LIN {X 0,Y 256.06,Z 399.2,A -85,B 0,C 180,E1 -18513.951,E2 -18513.951} C_VEL
LIN {X 0,Y 256.043,Z 399.215,A -85,B 0,C 180,E1 -18517.401,E2 -18517.401} C_VEL
LIN {X 0,Y 256.093,Z 399.188,A -85,B 0,C 180,E1 -18520.773,E2 -18520.773} C_VEL
LIN {X 0,Y 256.198,Z 399.177,A -85,B 0,C 180,E1 -18524.079,E2 -18524.079} C_VEL
LIN {X 0,Y 256.273,Z 399.171,A -85,B 0,C 180,E1 -18528.933,E2 -18528.933} C_VEL
LIN {X 0,Y 256.453,Z 399.151,A -85,B 0,C 180,E1 -18532.125,E2 -18532.125} C_VEL
LIN {X 0,Y 256.439,Z 399.144,A -85,B 0,C 180,E1 -18536.858,E2 -18536.858} C_VEL
LIN {X 0,Y 256.682,Z 399.137,A -85,B 0,C 180,E1 -18538.431,E2 -18538.431} C_VEL
LIN {X 0,Y 256.686,Z 399.109,A -85,B 0,C 180,E1 -18541.569,E2 -18541.569} C_VEL
LIN {X 0,Y 256.436,Z 399.14,A -85,B 0,C 180,E1 -18546.787,E2 -18546.787} C_VEL
LIN {X 0,Y 256.388,Z 399.171,A -85,B 0,C 180,E1 -18549.467,E2 -18549.467} C_VEL
LIN {X 0,Y 256.219,Z 399.192,A -85,B 0,C 180,E1 -18554.292,E2 -18554.292} C_VEL
LIN {X 0,Y 256.149,Z 399.182,A -85,B 0,C 180,E1 -18557.566,E2 -18557.566} C_VEL
LIN {X 0,Y 256.106,Z 399.186,A -85,B 0,C 180,E1 -18561.098,E2 -18561.098} C_VEL
LIN {X 0,Y 256.084,Z 399.409,A -85,B 0,C 180,E1 -18564.094,E2 -18564.094} C_VEL
LIN {X 0,Y 256.517,Z 400.923,A -85,B 0,C 180,E1 -18564.875,E2 -18564.875} C_VEL
LIN {X 0,Y 258.666,Z 404.243,A -85,B 0,C 180,E1 -18566.635,E2 -18566.635} C_VEL
LIN {X 0,Y 259.435,Z 406.128,A -85,B 0,C 180,E1 -18567.421,E2 -18567.421} C_VEL
LIN {X 0,Y 260.409,Z 407.557,A -85,B 0,C 180,E1 -18568.184,E2 -18568.184} C_VEL
LIN {X 0,Y 264.822,Z 416.275,A -85,B 0,C 180,E1 -18571.877,E2 -18571.877} C_VEL
LIN {X 0,Y 268.116,Z 423.333,A -85,B 0,C 180,E1 -18574.513,E2 -18574.513} C_VEL
LIN {X 0,Y 272.289,Z 433.348,A -85,B 0,C 180,E1 -18577.807,E2 -18577.807} C_VEL
LIN {X 0,Y 275.747,Z 442.564,A -85,B 0,C 180,E1 -18580.535,E2 -18580.535} C_VEL
LIN {X 0,Y 279.195,Z 452.902,A -85,B 0,C 180,E1 -18583.309,E2 -18583.309} C_VEL
LIN {X 0,Y 282.851,Z 466.067,A -85,B 0,C 180,E1 -18586.453,E2 -18586.453} C_VEL
LIN {X 0,Y 284.238,Z 471.069,A -85,B 0,C 180,E1 -18587.467,E2 -18587.467} C_VEL
LIN {X 0,Y 285.594,Z 474.475,A -85,B 0,C 180,E1 -18587.831,E2 -18587.831} C_VEL
LIN {X 0,Y 289.442,Z 502.295,A -85,B 0,C 180,E1 -18589.411,E2 -18589.411} C_VEL
LIN {X 0,Y 291.695,Z 522.529,A -85,B 0,C 180,E1 -18590.425,E2 -18590.425} C_VEL
LIN {X 0,Y 286.727,Z 629.994,A -85,B 0,C 180,E1 -18592.986,E2 -18592.986} C_VEL
LIN {X 0,Y 285.652,Z 646.755,A -85,B 0,C 180,E1 -18593.484,E2 -18593.484} C_VEL
LIN {X 0,Y 283.945,Z 662.444,A -85,B 0,C 180,E1 -18594.218,E2 -18594.218} C_VEL
LIN {X 0,Y 281.63,Z 677.308,A -85,B 0,C 180,E1 -18595.186,E2 -18595.186} C_VEL
LIN {X 0,Y 279.166,Z 690.887,A -85,B 0,C 180,E1 -18596.372,E2 -18596.372} C_VEL
LIN {X 0,Y 276.125,Z 704.824,A -85,B 0,C 180,E1 -18597.909,E2 -18597.909} C_VEL
LIN {X 0,Y 272.866,Z 717.487,A -85,B 0,C 180,E1 -18599.641,E2 -18599.641} C_VEL
LIN {X 0,Y 269.642,Z 729.09,A -85,B 0,C 180,E1 -18601.6,E2 -18601.6} C_VEL
LIN {X 0,Y 266.466,Z 740.121,A -85,B 0,C 180,E1 -18603.888,E2 -18603.888} C_VEL
LIN {X 0,Y 263.832,Z 748.759,A -85,B 0,C 180,E1 -18606.035,E2 -18606.035} C_VEL
LIN {X 0,Y 260.992,Z 757.604,A -85,B 0,C 180,E1 -18608.686,E2 -18608.686} C_VEL
LIN {X 0,Y 258.674,Z 765.048,A -85,B 0,C 180,E1 -18611.427,E2 -18611.427} C_VEL
LIN {X 0,Y 256.961,Z 770.984,A -85,B 0,C 180,E1 -18614.13,E2 -18614.13} C_VEL
LIN {X 0,Y 255.426,Z 776.513,A -85,B 0,C 180,E1 -18617.287,E2 -18617.287} C_VEL
LIN {X 0,Y 254.539,Z 780.689,A -85,B 0,C 180,E1 -18620.467,E2 -18620.467} C_VEL
LIN {X 0,Y 254.052,Z 783.623,A -85,B 0,C 180,E1 -18623.65,E2 -18623.65} C_VEL
LIN {X 0,Y 253.901,Z 785.384,A -85,B 0,C 180,E1 -18626.829,E2 -18626.829} C_VEL
LIN {X 0,Y 253.945,Z 785.994,A -85,B 0,C 180,E1 -18630.002,E2 -18630.002} C_VEL
LIN {X 0,Y 253.904,Z 785.421,A -85,B 0,C 180,E1 -18633.176,E2 -18633.176} C_VEL
LIN {X 0,Y 254.057,Z 783.708,A -85,B 0,C 180,E1 -18636.355,E2 -18636.355} C_VEL
LIN {X 0,Y 254.539,Z 780.819,A -85,B 0,C 180,E1 -18639.538,E2 -18639.538} C_VEL
LIN {X 0,Y 255.402,Z 776.687,A -85,B 0,C 180,E1 -18642.72,E2 -18642.72} C_VEL
LIN {X 0,Y 256.911,Z 771.213,A -85,B 0,C 180,E1 -18645.878,E2 -18645.878} C_VEL
LIN {X 0,Y 258.919,Z 764.244,A -85,B 0,C 180,E1 -18649.012,E2 -18649.012} C_VEL
LIN {X 0,Y 261.267,Z 756.773,A -85,B 0,C 180,E1 -18651.71,E2 -18651.71} C_VEL
LIN {X 0,Y 264.2,Z 747.772,A -85,B 0,C 180,E1 -18654.353,E2 -18654.353} C_VEL
LIN {X 0,Y 266.946,Z 738.581,A -85,B 0,C 180,E1 -18656.59,E2 -18656.59} C_VEL
LIN {X 0,Y 270.134,Z 727.708,A -85,B 0,C 180,E1 -18658.773,E2 -18658.773} C_VEL
LIN {X 0,Y 273.395,Z 715.822,A -85,B 0,C 180,E1 -18660.727,E2 -18660.727} C_VEL
LIN {X 0,Y 276.662,Z 702.814,A -85,B 0,C 180,E1 -18662.457,E2 -18662.457} C_VEL
LIN {X 0,Y 279.56,Z 689.399,A -85,B 0,C 180,E1 -18663.889,E2 -18663.889} C_VEL
LIN {X 0,Y 282.042,Z 675.326,A -85,B 0,C 180,E1 -18665.079,E2 -18665.079} C_VEL
LIN {X 0,Y 284.262,Z 660.41,A -85,B 0,C 180,E1 -18666.015,E2 -18666.015} C_VEL
LIN {X 0,Y 285.929,Z 644.861,A -85,B 0,C 180,E1 -18666.7,E2 -18666.7} C_VEL
LIN {X 0,Y 286.971,Z 626.833,A -85,B 0,C 180,E1 -18667.203,E2 -18667.203} C_VEL
LIN {X 0,Y 291.838,Z 522.454,A -85,B 0,C 180,E1 -18669.684,E2 -18669.684} C_VEL
LIN {X 0,Y 288.761,Z 496.622,A -85,B 0,C 180,E1 -18671.019,E2 -18671.019} C_VEL
LIN {X 0,Y 285.637,Z 474.073,A -85,B 0,C 180,E1 -18672.309,E2 -18672.309} C_VEL
LIN {X 0,Y 283.934,Z 470.142,A -85,B 0,C 180,E1 -18672.808,E2 -18672.808} C_VEL
LIN {X 0,Y 280.783,Z 458.187,A -85,B 0,C 180,E1 -18675.505,E2 -18675.505} C_VEL
LIN {X 0,Y 276.887,Z 445.879,A -85,B 0,C 180,E1 -18678.705,E2 -18678.705} C_VEL
LIN {X 0,Y 273.015,Z 434.978,A -85,B 0,C 180,E1 -18681.843,E2 -18681.843} C_VEL
LIN {X 0,Y 270.59,Z 428.968,A -85,B 0,C 180,E1 -18683.781,E2 -18683.781} C_VEL
LIN {X 0,Y 268.817,Z 426.664,A -85,B 0,C 180,E1 -18684.753,E2 -18684.753} C_VEL
LIN {X 0,Y 266.276,Z 425.384,A -85,B 0,C 180,E1 -18685.747,E2 -18685.747} C_VEL
LIN {X 0,Y 262.402,Z 425.077,A -85,B 0,C 180,E1 -18686.98,E2 -18686.98} C_VEL
LIN {X 0,Y 259.868,Z 425.572,A -85,B 0,C 180,E1 -18687.69,E2 -18687.69} C_VEL
LIN {X 0,Y 259.216,Z 426.104,A -85,B 0,C 180,E1 -18688.054,E2 -18688.054} C_VEL
LIN {X 0,Y 259.503,Z 427.426,A -85,B 0,C 180,E1 -18688.288,E2 -18688.288} C_VEL
LIN {X 0,Y 264.767,Z 441.663,A -85,B 0,C 180,E1 -18689.367,E2 -18689.367} C_VEL
LIN {X 0,Y 259.318,Z 542.125,A -85,B 0,C 180,E1 -18693.539,E2 -18693.539} C_VEL
LIN {X 0,Y 258.632,Z 557.649,A -85,B 0,C 180,E1 -18694.39,E2 -18694.39} C_VEL
LIN {X 0,Y 257.663,Z 572.895,A -85,B 0,C 180,E1 -18695.527,E2 -18695.527} C_VEL
LIN {X 0,Y 256.55,Z 586.386,A -85,B 0,C 180,E1 -18696.809,E2 -18696.809} C_VEL
LIN {X 0,Y 255.232,Z 601.418,A -85,B 0,C 180,E1 -18698.602,E2 -18698.602} C_VEL
LIN {X 0,Y 253.81,Z 615.052,A -85,B 0,C 180,E1 -18700.593,E2 -18700.593} C_VEL
LIN {X 0,Y 252.583,Z 627.546,A -85,B 0,C 180,E1 -18702.804,E2 -18702.804} C_VEL
LIN {X 0,Y 251.52,Z 637.995,A -85,B 0,C 180,E1 -18705.021,E2 -18705.021} C_VEL
LIN {X 0,Y 250.66,Z 647.631,A -85,B 0,C 180,E1 -18707.45,E2 -18707.45} C_VEL
LIN {X 0,Y 249.954,Z 656.985,A -85,B 0,C 180,E1 -18710.287,E2 -18710.287} C_VEL
LIN {X 0,Y 249.49,Z 663.619,A -85,B 0,C 180,E1 -18712.717,E2 -18712.717} C_VEL
LIN {X 0,Y 249.243,Z 670.808,A -85,B 0,C 180,E1 -18715.958,E2 -18715.958} C_VEL
LIN {X 0,Y 249.469,Z 676.374,A -85,B 0,C 180,E1 -18719.193,E2 -18719.193} C_VEL
LIN {X 0,Y 250.022,Z 679.487,A -85,B 0,C 180,E1 -18721.611,E2 -18721.611} C_VEL
LIN {X 0,Y 251.132,Z 682.416,A -85,B 0,C 180,E1 -18724.816,E2 -18724.816} C_VEL
LIN {X 0,Y 252.623,Z 684.009,A -85,B 0,C 180,E1 -18727.996,E2 -18727.996} C_VEL
LIN {X 0,Y 254.788,Z 684.233,A -85,B 0,C 180,E1 -18731.133,E2 -18731.133} C_VEL
LIN {X 0,Y 257.49,Z 683.132,A -85,B 0,C 180,E1 -18734.22,E2 -18734.22} C_VEL
LIN {X 0,Y 260.989,Z 680.652,A -85,B 0,C 180,E1 -18737.23,E2 -18737.23} C_VEL
LIN {X 0,Y 264.933,Z 676.843,A -85,B 0,C 180,E1 -18740.173,E2 -18740.173} C_VEL
LIN {X 0,Y 269.585,Z 671.523,A -85,B 0,C 180,E1 -18743.019,E2 -18743.019} C_VEL
LIN {X 0,Y 274.771,Z 664.681,A -85,B 0,C 180,E1 -18745.774,E2 -18745.774} C_VEL
LIN {X 0,Y 279.832,Z 657.27,A -85,B 0,C 180,E1 -18748.093,E2 -18748.093} C_VEL
LIN {X 0,Y 286.156,Z 647.005,A -85,B 0,C 180,E1 -18750.638,E2 -18750.638} C_VEL
LIN {X 0,Y 292.113,Z 636.101,A -85,B 0,C 180,E1 -18752.774,E2 -18752.774} C_VEL
LIN {X 0,Y 298.05,Z 624.066,A -85,B 0,C 180,E1 -18754.671,E2 -18754.671} C_VEL
LIN {X 0,Y 302.909,Z 613.048,A -85,B 0,C 180,E1 -18756.068,E2 -18756.068} C_VEL
LIN {X 0,Y 308.468,Z 598.622,A -85,B 0,C 180,E1 -18757.55,E2 -18757.55} C_VEL
LIN {X 0,Y 312.634,Z 585.97,A -85,B 0,C 180,E1 -18758.595,E2 -18758.595} C_VEL
LIN {X 0,Y 317.001,Z 569.833,A -85,B 0,C 180,E1 -18759.649,E2 -18759.649} C_VEL
LIN {X 0,Y 321.934,Z 549.906,A -85,B 0,C 180,E1 -18760.655,E2 -18760.655} C_VEL
LIN {X 0,Y 331.491,Z 513.679,A -85,B 0,C 180,E1 -18762.202,E2 -18762.202} C_VEL
LIN {X 0,Y 331.324,Z 514.505,A -85,B 0,C 180,E1 -18763.011,E2 -18763.011} C_VEL
LIN {X 0,Y 328.78,Z 524.894,A -85,B 0,C 180,E1 -18763.854,E2 -18763.854} C_VEL
LIN {X 0,Y 327.692,Z 529.255,A -85,B 0,C 180,E1 -18764.081,E2 -18764.081} C_VEL
LIN {X 0,Y 312.213,Z 593.031,A -85,B 0,C 180,E1 -18766.639,E2 -18766.639} C_VEL
LIN {X 0,Y 306.727,Z 610.777,A -85,B 0,C 180,E1 -18767.503,E2 -18767.503} C_VEL
LIN {X 0,Y 300.345,Z 628.134,A -85,B 0,C 180,E1 -18768.618,E2 -18768.618} C_VEL
LIN {X 0,Y 293.51,Z 644.352,A -85,B 0,C 180,E1 -18769.944,E2 -18769.944} C_VEL
LIN {X 0,Y 286.435,Z 659.292,A -85,B 0,C 180,E1 -18771.491,E2 -18771.491} C_VEL
LIN {X 0,Y 279.486,Z 673.037,A -85,B 0,C 180,E1 -18773.327,E2 -18773.327} C_VEL
LIN {X 0,Y 274.434,Z 683.089,A -85,B 0,C 180,E1 -18774.938,E2 -18774.938} C_VEL
LIN {X 0,Y 271.434,Z 697.667,A -85,B 0,C 180,E1 -18776.394,E2 -18776.394} C_VEL
LIN {X 0,Y 268.34,Z 710.262,A -85,B 0,C 180,E1 -18777.968,E2 -18777.968} C_VEL
LIN {X 0,Y 264.895,Z 722.987,A -85,B 0,C 180,E1 -18779.946,E2 -18779.946} C_VEL
LIN {X 0,Y 261.612,Z 733.628,A -85,B 0,C 180,E1 -18781.955,E2 -18781.955} C_VEL
LIN {X 0,Y 258.634,Z 743.458,A -85,B 0,C 180,E1 -18784.227,E2 -18784.227} C_VEL
LIN {X 0,Y 255.453,Z 753.06,A -85,B 0,C 180,E1 -18786.916,E2 -18786.916} C_VEL
LIN {X 0,Y 252.869,Z 761.05,A -85,B 0,C 180,E1 -18789.669,E2 -18789.669} C_VEL
LIN {X 0,Y 250.628,Z 768.04,A -85,B 0,C 180,E1 -18792.642,E2 -18792.642} C_VEL
LIN {X 0,Y 248.854,Z 774.37,A -85,B 0,C 180,E1 -18796.108,E2 -18796.108} C_VEL
LIN {X 0,Y 247.978,Z 777.851,A -85,B 0,C 180,E1 -18798.555,E2 -18798.555} C_VEL
LIN {X 0,Y 247.273,Z 781.385,A -85,B 0,C 180,E1 -18801.828,E2 -18801.828} C_VEL
LIN {X 0,Y 246.97,Z 783.705,A -85,B 0,C 180,E1 -18805.1,E2 -18805.1} C_VEL
LIN {X 0,Y 246.925,Z 784.867,A -85,B 0,C 180,E1 -18808.367,E2 -18808.367} C_VEL
LIN {X 0,Y 246.956,Z 785.018,A -85,B 0,C 180,E1 -18809.997,E2 -18809.997} C_VEL
LIN {X 0,Y 246.896,Z 784.418,A -85,B 0,C 180,E1 -18813.261,E2 -18813.261} C_VEL
LIN {X 0,Y 247.062,Z 782.669,A -85,B 0,C 180,E1 -18816.531,E2 -18816.531} C_VEL
LIN {X 0,Y 247.553,Z 779.742,A -85,B 0,C 180,E1 -18819.805,E2 -18819.805} C_VEL
LIN {X 0,Y 248.46,Z 775.566,A -85,B 0,C 180,E1 -18823.076,E2 -18823.076} C_VEL
LIN {X 0,Y 250.017,Z 770.028,A -85,B 0,C 180,E1 -18826.323,E2 -18826.323} C_VEL
LIN {X 0,Y 252.163,Z 762.976,A -85,B 0,C 180,E1 -18829.536,E2 -18829.536} C_VEL
LIN {X 0,Y 254.637,Z 755.417,A -85,B 0,C 180,E1 -18832.3,E2 -18832.3} C_VEL
LIN {X 0,Y 257.243,Z 747.712,A -85,B 0,C 180,E1 -18834.619,E2 -18834.619} C_VEL
LIN {X 0,Y 260.039,Z 738.343,A -85,B 0,C 180,E1 -18836.991,E2 -18836.991} C_VEL
LIN {X 0,Y 263.302,Z 727.905,A -85,B 0,C 180,E1 -18839.149,E2 -18839.149} C_VEL
LIN {X 0,Y 266.65,Z 716.184,A -85,B 0,C 180,E1 -18841.145,E2 -18841.145} C_VEL
LIN {X 0,Y 269.966,Z 703.349,A -85,B 0,C 180,E1 -18842.915,E2 -18842.915} C_VEL
LIN {X 0,Y 273.122,Z 689.158,A -85,B 0,C 180,E1 -18844.476,E2 -18844.476} C_VEL
LIN {X 0,Y 275.676,Z 675.29,A -85,B 0,C 180,E1 -18845.67,E2 -18845.67} C_VEL
LIN {X 0,Y 277.888,Z 660.441,A -85,B 0,C 180,E1 -18846.631,E2 -18846.631} C_VEL
LIN {X 0,Y 279.595,Z 644.94,A -85,B 0,C 180,E1 -18847.327,E2 -18847.327} C_VEL
LIN {X 0,Y 280.717,Z 627.069,A -85,B 0,C 180,E1 -18847.831,E2 -18847.831} C_VEL
LIN {X 0,Y 284.46,Z 548.125,A -85,B 0,C 180,E1 -18849.738,E2 -18849.738} C_VEL
LIN {X 0,Y 285.859,Z 517.692,A -85,B 0,C 180,E1 -18850.481,E2 -18850.481} C_VEL
LIN {X 0,Y 282.554,Z 482.323,A -85,B 0,C 180,E1 -18852.235,E2 -18852.235} C_VEL
LIN {X 0,Y 281.195,Z 470.402,A -85,B 0,C 180,E1 -18852.893,E2 -18852.893} C_VEL
LIN {X 0,Y 279.904,Z 467.147,A -85,B 0,C 180,E1 -18853.269,E2 -18853.269} C_VEL
LIN {X 0,Y 274.249,Z 446.451,A -85,B 0,C 180,E1 -18856.798,E2 -18856.798} C_VEL
LIN {X 0,Y 271.321,Z 436.268,A -85,B 0,C 180,E1 -18858.689,E2 -18858.689} C_VEL
LIN {X 0,Y 267.713,Z 429.764,A -85,B 0,C 180,E1 -18860.461,E2 -18860.461} C_VEL
LIN {X 0,Y 261.581,Z 419.504,A -85,B 0,C 180,E1 -18863.766,E2 -18863.766} C_VEL
LIN {X 0,Y 255.88,Z 410.717,A -85,B 0,C 180,E1 -18867.171,E2 -18867.171} C_VEL
LIN {X 0,Y 253.967,Z 408.628,A -85,B 0,C 180,E1 -18868.279,E2 -18868.279} C_VEL
LIN {X 0,Y 251.92,Z 404.976,A -85,B 0,C 180,E1 -18869.857,E2 -18869.857} C_VEL
LIN {X 0,Y 250.549,Z 403.702,A -85,B 0,C 180,E1 -18870.738,E2 -18870.738} C_VEL
LIN {X 0,Y 249.097,Z 400.489,A -85,B 0,C 180,E1 -18872.256,E2 -18872.256} C_VEL
LIN {X 0,Y 249.007,Z 400.094,A -85,B 0,C 180,E1 -18873.155,E2 -18873.155} C_VEL
LIN {X 0,Y 248.992,Z 400.081,A -85,B 0,C 180,E1 -18876.724,E2 -18876.724} C_VEL
LIN {X 0,Y 249.028,Z 400.066,A -85,B 0,C 180,E1 -18880.205,E2 -18880.205} C_VEL
LIN {X 0,Y 249.144,Z 400.06,A -85,B 0,C 180,E1 -18883.615,E2 -18883.615} C_VEL
LIN {X 0,Y 249.215,Z 400.055,A -85,B 0,C 180,E1 -18888.615,E2 -18888.615} C_VEL
LIN {X 0,Y 249.403,Z 400.025,A -85,B 0,C 180,E1 -18891.9,E2 -18891.9} C_VEL
LIN {X 0,Y 249.249,Z 400.035,A -85,B 0,C 180,E1 -18895.148,E2 -18895.148} C_VEL
LIN {X 0,Y 249.643,Z 400.013,A -85,B 0,C 180,E1 -18898.387,E2 -18898.387} C_VEL
LIN {X 0,Y 249.647,Z 399.986,A -85,B 0,C 180,E1 -18901.613,E2 -18901.613} C_VEL
LIN {X 0,Y 249.405,Z 400.016,A -85,B 0,C 180,E1 -18906.773,E2 -18906.773} C_VEL
LIN {X 0,Y 249.319,Z 400.045,A -85,B 0,C 180,E1 -18909.738,E2 -18909.738} C_VEL
LIN {X 0,Y 249.159,Z 400.065,A -85,B 0,C 180,E1 -18914.706,E2 -18914.706} C_VEL
LIN {X 0,Y 249.082,Z 400.067,A -85,B 0,C 180,E1 -18918.082,E2 -18918.082} C_VEL
LIN {X 0,Y 249.083,Z 400.216,A -85,B 0,C 180,E1 -18921.043,E2 -18921.043} C_VEL
LIN {X 0,Y 249.188,Z 400.824,A -85,B 0,C 180,E1 -18921.509,E2 -18921.509} C_VEL
LIN {X 0,Y 250.597,Z 403.746,A -85,B 0,C 180,E1 -18923.118,E2 -18923.118} C_VEL
LIN {X 0,Y 251.593,Z 404.822,A -85,B 0,C 180,E1 -18923.894,E2 -18923.894} C_VEL
LIN {X 0,Y 254.111,Z 409.478,A -85,B 0,C 180,E1 -18926.265,E2 -18926.265} C_VEL
LIN {X 0,Y 258.474,Z 418.037,A -85,B 0,C 180,E1 -18930.2,E2 -18930.2} C_VEL
LIN {X 0,Y 263.14,Z 428.048,A -85,B 0,C 180,E1 -18934.116,E2 -18934.116} C_VEL
LIN {X 0,Y 267.456,Z 438.688,A -85,B 0,C 180,E1 -18937.693,E2 -18937.693} C_VEL
LIN {X 0,Y 270.786,Z 447.921,A -85,B 0,C 180,E1 -18940.455,E2 -18940.455} C_VEL
LIN {X 0,Y 274.147,Z 458.426,A -85,B 0,C 180,E1 -18943.274,E2 -18943.274} C_VEL
LIN {X 0,Y 277.343,Z 470.167,A -85,B 0,C 180,E1 -18946.078,E2 -18946.078} C_VEL
LIN {X 0,Y 280.543,Z 477.276,A -85,B 0,C 180,E1 -18946.99,E2 -18946.99} C_VEL
LIN {X 0,Y 284.15,Z 504.547,A -85,B 0,C 180,E1 -18948.568,E2 -18948.568} C_VEL
LIN {X 0,Y 286.198,Z 522.329,A -85,B 0,C 180,E1 -18949.506,E2 -18949.506} C_VEL
LIN {X 0,Y 281.833,Z 615.616,A -85,B 0,C 180,E1 -18951.779,E2 -18951.779} C_VEL
LIN {X 0,Y 280.282,Z 643.468,A -85,B 0,C 180,E1 -18952.497,E2 -18952.497} C_VEL
LIN {X 0,Y 278.73,Z 658.745,A -85,B 0,C 180,E1 -18953.16,E2 -18953.16} C_VEL
LIN {X 0,Y 276.385,Z 674.078,A -85,B 0,C 180,E1 -18954.099,E2 -18954.099} C_VEL
LIN {X 0,Y 273.698,Z 688.704,A -85,B 0,C 180,E1 -18955.327,E2 -18955.327} C_VEL
LIN {X 0,Y 270.856,Z 702.005,A -85,B 0,C 180,E1 -18956.764,E2 -18956.764} C_VEL
LIN {X 0,Y 267.417,Z 715.161,A -85,B 0,C 180,E1 -18958.514,E2 -18958.514} C_VEL
LIN {X 0,Y 263.996,Z 727.151,A -85,B 0,C 180,E1 -18960.498,E2 -18960.498} C_VEL
LIN {X 0,Y 260.683,Z 738.108,A -85,B 0,C 180,E1 -18962.724,E2 -18962.724} C_VEL
LIN {X 0,Y 257.8,Z 747.34,A -85,B 0,C 180,E1 -18965.007,E2 -18965.007} C_VEL
LIN {X 0,Y 254.705,Z 756.407,A -85,B 0,C 180,E1 -18967.706,E2 -18967.706} C_VEL
LIN {X 0,Y 252.24,Z 763.938,A -85,B 0,C 180,E1 -18970.47,E2 -18970.47} C_VEL
LIN {X 0,Y 250.089,Z 770.97,A -85,B 0,C 180,E1 -18973.682,E2 -18973.682} C_VEL
LIN {X 0,Y 248.458,Z 776.499,A -85,B 0,C 180,E1 -18976.924,E2 -18976.924} C_VEL
LIN {X 0,Y 247.515,Z 780.675,A -85,B 0,C 180,E1 -18980.194,E2 -18980.194} C_VEL
LIN {X 0,Y 246.973,Z 783.609,A -85,B 0,C 180,E1 -18983.467,E2 -18983.467} C_VEL
LIN {X 0,Y 246.806,Z 785.37,A -85,B 0,C 180,E1 -18986.738,E2 -18986.738} C_VEL
LIN {X 0,Y 246.857,Z 785.981,A -85,B 0,C 180,E1 -18990.003,E2 -18990.003} C_VEL
LIN {X 0,Y 246.809,Z 785.407,A -85,B 0,C 180,E1 -18993.267,E2 -18993.267} C_VEL
LIN {X 0,Y 246.976,Z 783.694,A -85,B 0,C 180,E1 -18996.538,E2 -18996.538} C_VEL
LIN {X 0,Y 247.514,Z 780.804,A -85,B 0,C 180,E1 -18999.812,E2 -18999.812} C_VEL
LIN {X 0,Y 248.437,Z 776.671,A -85,B 0,C 180,E1 -19003.082,E2 -19003.082} C_VEL
LIN {X 0,Y 250.038,Z 771.196,A -85,B 0,C 180,E1 -19006.327,E2 -19006.327} C_VEL
LIN {X 0,Y 252.157,Z 764.226,A -85,B 0,C 180,E1 -19009.542,E2 -19009.542} C_VEL
LIN {X 0,Y 254.635,Z 756.754,A -85,B 0,C 180,E1 -19012.305,E2 -19012.305} C_VEL
LIN {X 0,Y 257.692,Z 747.751,A -85,B 0,C 180,E1 -19015.009,E2 -19015.009} C_VEL
LIN {X 0,Y 260.553,Z 738.559,A -85,B 0,C 180,E1 -19017.296,E2 -19017.296} C_VEL
LIN {X 0,Y 264.233,Z 726.718,A -85,B 0,C 180,E1 -19019.697,E2 -19019.697} C_VEL
LIN {X 0,Y 267.597,Z 714.638,A -85,B 0,C 180,E1 -19021.689,E2 -19021.689} C_VEL
LIN {X 0,Y 271.082,Z 701.373,A -85,B 0,C 180,E1 -19023.432,E2 -19023.432} C_VEL
LIN {X 0,Y 274.096,Z 687.306,A -85,B 0,C 180,E1 -19024.921,E2 -19024.921} C_VEL
LIN {X 0,Y 276.632,Z 673.05,A -85,B 0,C 180,E1 -19026.095,E2 -19026.095} C_VEL
LIN {X 0,Y 278.867,Z 658.087,A -85,B 0,C 180,E1 -19026.994,E2 -19026.994} C_VEL
LIN {X 0,Y 280.467,Z 642.428,A -85,B 0,C 180,E1 -19027.649,E2 -19027.649} C_VEL
LIN {X 0,Y 282.387,Z 605.812,A -85,B 0,C 180,E1 -19028.575,E2 -19028.575} C_VEL
LIN {X 0,Y 286.277,Z 522.1,A -85,B 0,C 180,E1 -19030.62,E2 -19030.62} C_VEL
LIN {X 0,Y 282.056,Z 487.271,A -85,B 0,C 180,E1 -19032.523,E2 -19032.523} C_VEL
LIN {X 0,Y 280.463,Z 476.976,A -85,B 0,C 180,E1 -19033.173,E2 -19033.173} C_VEL
LIN {X 0,Y 277.442,Z 470.311,A -85,B 0,C 180,E1 -19034.025,E2 -19034.025} C_VEL
LIN {X 0,Y 274.375,Z 459.224,A -85,B 0,C 180,E1 -19036.669,E2 -19036.669} C_VEL
LIN {X 0,Y 270.712,Z 447.562,A -85,B 0,C 180,E1 -19039.804,E2 -19039.804} C_VEL
LIN {X 0,Y 267.162,Z 437.743,A -85,B 0,C 180,E1 -19042.768,E2 -19042.768} C_VEL
LIN {X 0,Y 262.413,Z 426.238,A -85,B 0,C 180,E1 -19046.699,E2 -19046.699} C_VEL
LIN {X 0,Y 260.923,Z 425.262,A -85,B 0,C 180,E1 -19047.404,E2 -19047.404} C_VEL
LIN {X 0,Y 259.868,Z 425.572,A -85,B 0,C 180,E1 -19047.69,E2 -19047.69} C_VEL
LIN {X 0,Y 258.728,Z 426.728,A -85,B 0,C 180,E1 -19048.002,E2 -19048.002} C_VEL
LIN {X 0,Y 257.868,Z 429.291,A -85,B 0,C 180,E1 -19048.232,E2 -19048.232} C_VEL
LIN {X 0,Y 256.042,Z 445.528,A -85,B 0,C 180,E1 -19048.874,E2 -19048.874} C_VEL
LIN {X 0,Y 256.872,Z 453.057,A -85,B 0,C 180,E1 -19049.278,E2 -19049.278} C_VEL
LIN {X 0,Y 257.239,Z 456.327,A -85,B 0,C 180,E1 -19049.478,E2 -19049.478} C_VEL
LIN {X 0,Y 252.462,Z 540.302,A -85,B 0,C 180,E1 -19053.1,E2 -19053.1} C_VEL
LIN {X 0,Y 251.736,Z 557.141,A -85,B 0,C 180,E1 -19054.026,E2 -19054.026} C_VEL
LIN {X 0,Y 250.689,Z 573.249,A -85,B 0,C 180,E1 -19055.243,E2 -19055.243} C_VEL
LIN {X 0,Y 249.548,Z 586.854,A -85,B 0,C 180,E1 -19056.559,E2 -19056.559} C_VEL
LIN {X 0,Y 248.347,Z 600.512,A -85,B 0,C 180,E1 -19058.196,E2 -19058.196} C_VEL
LIN {X 0,Y 246.859,Z 614.452,A -85,B 0,C 180,E1 -19060.24,E2 -19060.24} C_VEL
LIN {X 0,Y 245.604,Z 627.238,A -85,B 0,C 180,E1 -19062.515,E2 -19062.515} C_VEL
LIN {X 0,Y 244.42,Z 638.824,A -85,B 0,C 180,E1 -19065.002,E2 -19065.002} C_VEL
LIN {X 0,Y 243.546,Z 648.466,A -85,B 0,C 180,E1 -19067.501,E2 -19067.501} C_VEL
LIN {X 0,Y 242.832,Z 657.835,A -85,B 0,C 180,E1 -19070.42,E2 -19070.42} C_VEL
LIN {X 0,Y 242.343,Z 664.555,A -85,B 0,C 180,E1 -19072.92,E2 -19072.92} C_VEL
LIN {X 0,Y 242.164,Z 671.032,A -85,B 0,C 180,E1 -19075.839,E2 -19075.839} C_VEL
LIN {X 0,Y 242.407,Z 676.813,A -85,B 0,C 180,E1 -19079.169,E2 -19079.169} C_VEL
LIN {X 0,Y 242.962,Z 680.174,A -85,B 0,C 180,E1 -19081.657,E2 -19081.657} C_VEL
LIN {X 0,Y 244.127,Z 683.358,A -85,B 0,C 180,E1 -19084.954,E2 -19084.954} C_VEL
LIN {X 0,Y 245.71,Z 685.199,A -85,B 0,C 180,E1 -19088.222,E2 -19088.222} C_VEL
LIN {X 0,Y 247.987,Z 685.685,A -85,B 0,C 180,E1 -19091.442,E2 -19091.442} C_VEL
LIN {X 0,Y 250.842,Z 684.865,A -85,B 0,C 180,E1 -19094.605,E2 -19094.605} C_VEL
LIN {X 0,Y 254.5,Z 682.691,A -85,B 0,C 180,E1 -19097.684,E2 -19097.684} C_VEL
LIN {X 0,Y 258.659,Z 679.212,A -85,B 0,C 180,E1 -19100.684,E2 -19100.684} C_VEL
LIN {X 0,Y 263.551,Z 674.306,A -85,B 0,C 180,E1 -19103.578,E2 -19103.578} C_VEL
LIN {X 0,Y 268.993,Z 667.947,A -85,B 0,C 180,E1 -19106.37,E2 -19106.37} C_VEL
LIN {X 0,Y 274.284,Z 660.999,A -85,B 0,C 180,E1 -19108.714,E2 -19108.714} C_VEL
LIN {X 0,Y 280.936,Z 651.283,A -85,B 0,C 180,E1 -19111.271,E2 -19111.271} C_VEL
LIN {X 0,Y 287.127,Z 641.165,A -85,B 0,C 180,E1 -19113.417,E2 -19113.417} C_VEL
LIN {X 0,Y 293.803,Z 628.999,A -85,B 0,C 180,E1 -19115.456,E2 -19115.456} C_VEL
LIN {X 0,Y 299.892,Z 616.516,A -85,B 0,C 180,E1 -19117.117,E2 -19117.117} C_VEL
LIN {X 0,Y 305.701,Z 602.96,A -85,B 0,C 180,E1 -19118.558,E2 -19118.558} C_VEL
LIN {X 0,Y 310.664,Z 589.242,A -85,B 0,C 180,E1 -19119.723,E2 -19119.723} C_VEL
LIN {X 0,Y 315.404,Z 573.289,A -85,B 0,C 180,E1 -19120.78,E2 -19120.78} C_VEL
LIN {X 0,Y 320.479,Z 554.01,A -85,B 0,C 180,E1 -19121.769,E2 -19121.769} C_VEL
LIN {X 0,Y 327.218,Z 529.505,A -85,B 0,C 180,E1 -19122.819,E2 -19122.819} C_VEL
LIN {X 0,Y 311.354,Z 590.804,A -85,B 0,C 180,E1 -19125.251,E2 -19125.251} C_VEL
LIN {X 0,Y 305.402,Z 608.987,A -85,B 0,C 180,E1 -19126.11,E2 -19126.11} C_VEL
LIN {X 0,Y 298.793,Z 625.943,A -85,B 0,C 180,E1 -19127.167,E2 -19127.167} C_VEL
LIN {X 0,Y 292.154,Z 640.904,A -85,B 0,C 180,E1 -19128.351,E2 -19128.351} C_VEL
LIN {X 0,Y 285.386,Z 654.562,A -85,B 0,C 180,E1 -19129.678,E2 -19129.678} C_VEL
LIN {X 0,Y 278.323,Z 667.81,A -85,B 0,C 180,E1 -19131.318,E2 -19131.318} C_VEL
LIN {X 0,Y 270.965,Z 680.883,A -85,B 0,C 180,E1 -19133.374,E2 -19133.374} C_VEL
LIN {X 0,Y 268.125,Z 685.932,A -85,B 0,C 180,E1 -19134.316,E2 -19134.316} C_VEL
LIN {X 0,Y 264.818,Z 700.803,A -85,B 0,C 180,E1 -19135.903,E2 -19135.903} C_VEL
LIN {X 0,Y 261.311,Z 714.049,A -85,B 0,C 180,E1 -19137.685,E2 -19137.685} C_VEL
LIN {X 0,Y 257.763,Z 726.132,A -85,B 0,C 180,E1 -19139.705,E2 -19139.705} C_VEL
LIN {X 0,Y 254.235,Z 737.153,A -85,B 0,C 180,E1 -19141.967,E2 -19141.967} C_VEL
LIN {X 0,Y 251.268,Z 746.429,A -85,B 0,C 180,E1 -19144.305,E2 -19144.305} C_VEL
LIN {X 0,Y 248.082,Z 755.527,A -85,B 0,C 180,E1 -19147.072,E2 -19147.072} C_VEL
LIN {X 0,Y 245.467,Z 763.071,A -85,B 0,C 180,E1 -19149.903,E2 -19149.903} C_VEL
LIN {X 0,Y 243.677,Z 768.433,A -85,B 0,C 180,E1 -19152.334,E2 -19152.334} C_VEL
LIN {X 0,Y 241.93,Z 774.386,A -85,B 0,C 180,E1 -19155.702,E2 -19155.702} C_VEL
LIN {X 0,Y 240.971,Z 777.867,A -85,B 0,C 180,E1 -19158.217,E2 -19158.217} C_VEL
LIN {X 0,Y 240.213,Z 781.4,A -85,B 0,C 180,E1 -19161.586,E2 -19161.586} C_VEL
LIN {X 0,Y 239.864,Z 783.74,A -85,B 0,C 180,E1 -19164.999,E2 -19164.999} C_VEL
LIN {X 0,Y 239.836,Z 784.881,A -85,B 0,C 180,E1 -19168.318,E2 -19168.318} C_VEL
LIN {X 0,Y 239.866,Z 785.032,A -85,B 0,C 180,E1 -19169.997,E2 -19169.997} C_VEL
LIN {X 0,Y 239.8,Z 784.432,A -85,B 0,C 180,E1 -19173.358,E2 -19173.358} C_VEL
LIN {X 0,Y 239.985,Z 782.682,A -85,B 0,C 180,E1 -19176.724,E2 -19176.724} C_VEL
LIN {X 0,Y 240.508,Z 779.756,A -85,B 0,C 180,E1 -19180.095,E2 -19180.095} C_VEL
LIN {X 0,Y 241.509,Z 775.58,A -85,B 0,C 180,E1 -19183.459,E2 -19183.459} C_VEL
LIN {X 0,Y 243.17,Z 770.042,A -85,B 0,C 180,E1 -19186.796,E2 -19186.796} C_VEL
LIN {X 0,Y 245.426,Z 762.991,A -85,B 0,C 180,E1 -19190.095,E2 -19190.095} C_VEL
LIN {X 0,Y 248.027,Z 755.432,A -85,B 0,C 180,E1 -19192.928,E2 -19192.928} C_VEL
LIN {X 0,Y 251.225,Z 746.319,A -85,B 0,C 180,E1 -19195.694,E2 -19195.694} C_VEL
LIN {X 0,Y 253.581,Z 738.693,A -85,B 0,C 180,E1 -19197.644,E2 -19197.644} C_VEL
LIN {X 0,Y 257.077,Z 727.923,A -85,B 0,C 180,E1 -19199.925,E2 -19199.925} C_VEL
LIN {X 0,Y 260.59,Z 716.204,A -85,B 0,C 180,E1 -19201.953,E2 -19201.953} C_VEL
LIN {X 0,Y 264.017,Z 703.373,A -85,B 0,C 180,E1 -19203.754,E2 -19203.754} C_VEL
LIN {X 0,Y 267.293,Z 689.186,A -85,B 0,C 180,E1 -19205.338,E2 -19205.338} C_VEL
LIN {X 0,Y 269.934,Z 675.324,A -85,B 0,C 180,E1 -19206.55,E2 -19206.55} C_VEL
LIN {X 0,Y 272.236,Z 660.487,A -85,B 0,C 180,E1 -19207.52,E2 -19207.52} C_VEL
LIN {X 0,Y 274.004,Z 645.006,A -85,B 0,C 180,E1 -19208.224,E2 -19208.224} C_VEL
LIN {X 0,Y 275.24,Z 625.382,A -85,B 0,C 180,E1 -19208.78,E2 -19208.78} C_VEL
LIN {X 0,Y 279.051,Z 548.23,A -85,B 0,C 180,E1 -19210.667,E2 -19210.667} C_VEL
LIN {X 0,Y 280.409,Z 518.014,A -85,B 0,C 180,E1 -19211.431,E2 -19211.431} C_VEL
LIN {X 0,Y 277.415,Z 484.564,A -85,B 0,C 180,E1 -19213.132,E2 -19213.132} C_VEL
LIN {X 0,Y 276.165,Z 473.338,A -85,B 0,C 180,E1 -19213.771,E2 -19213.771} C_VEL
LIN {X 0,Y 273.569,Z 466.667,A -85,B 0,C 180,E1 -19214.602,E2 -19214.602} C_VEL
LIN {X 0,Y 268.363,Z 446.983,A -85,B 0,C 180,E1 -19218.131,E2 -19218.131} C_VEL
LIN {X 0,Y 266.728,Z 440.891,A -85,B 0,C 180,E1 -19219.297,E2 -19219.297} C_VEL
LIN {X 0,Y 263.136,Z 434.419,A -85,B 0,C 180,E1 -19221.123,E2 -19221.123} C_VEL
LIN {X 0,Y 257.763,Z 425.318,A -85,B 0,C 180,E1 -19224.112,E2 -19224.112} C_VEL
LIN {X 0,Y 251.565,Z 415.797,A -85,B 0,C 180,E1 -19227.94,E2 -19227.94} C_VEL
LIN {X 0,Y 250.342,Z 414.428,A -85,B 0,C 180,E1 -19228.711,E2 -19228.711} C_VEL
LIN {X 0,Y 248.682,Z 411.389,A -85,B 0,C 180,E1 -19230.039,E2 -19230.039} C_VEL
LIN {X 0,Y 246.15,Z 408.129,A -85,B 0,C 180,E1 -19231.895,E2 -19231.895} C_VEL
LIN {X 0,Y 245.322,Z 406.223,A -85,B 0,C 180,E1 -19232.718,E2 -19232.718} C_VEL
LIN {X 0,Y 243.262,Z 404.225,A -85,B 0,C 180,E1 -19234.319,E2 -19234.319} C_VEL
LIN {X 0,Y 242.003,Z 401.325,A -85,B 0,C 180,E1 -19236.01,E2 -19236.01} C_VEL
LIN {X 0,Y 241.961,Z 400.969,A -85,B 0,C 180,E1 -19236.914,E2 -19236.914} C_VEL
LIN {X 0,Y 242.004,Z 400.948,A -85,B 0,C 180,E1 -19241.371,E2 -19241.371} C_VEL
LIN {X 0,Y 242.092,Z 400.928,A -85,B 0,C 180,E1 -19244.855,E2 -19244.855} C_VEL
LIN {X 0,Y 242.328,Z 400.896,A -85,B 0,C 180,E1 -19250.404,E2 -19250.404} C_VEL
LIN {X 0,Y 242.381,Z 400.916,A -85,B 0,C 180,E1 -19253.34,E2 -19253.34} C_VEL
LIN {X 0,Y 242.603,Z 400.89,A -85,B 0,C 180,E1 -19258.34,E2 -19258.34} C_VEL
LIN {X 0,Y 242.607,Z 400.862,A -85,B 0,C 180,E1 -19261.66,E2 -19261.66} C_VEL
LIN {X 0,Y 242.385,Z 400.889,A -85,B 0,C 180,E1 -19266.747,E2 -19266.747} C_VEL
LIN {X 0,Y 242.247,Z 400.92,A -85,B 0,C 180,E1 -19270.025,E2 -19270.025} C_VEL
LIN {X 0,Y 242.109,Z 400.935,A -85,B 0,C 180,E1 -19275.145,E2 -19275.145} C_VEL
LIN {X 0,Y 242.095,Z 401.169,A -85,B 0,C 180,E1 -19277.529,E2 -19277.529} C_VEL
LIN {X 0,Y 243.163,Z 404.035,A -85,B 0,C 180,E1 -19279.413,E2 -19279.413} C_VEL
LIN {X 0,Y 244.696,Z 405.743,A -85,B 0,C 180,E1 -19280.871,E2 -19280.871} C_VEL
LIN {X 0,Y 246.143,Z 409.018,A -85,B 0,C 180,E1 -19282.672,E2 -19282.672} C_VEL
LIN {X 0,Y 247.078,Z 410.158,A -85,B 0,C 180,E1 -19283.467,E2 -19283.467} C_VEL
LIN {X 0,Y 249.561,Z 414.719,A -85,B 0,C 180,E1 -19285.88,E2 -19285.88} C_VEL
LIN {X 0,Y 253.838,Z 423.22,A -85,B 0,C 180,E1 -19289.892,E2 -19289.892} C_VEL
LIN {X 0,Y 258.102,Z 432.585,A -85,B 0,C 180,E1 -19293.651,E2 -19293.651} C_VEL
LIN {X 0,Y 262.577,Z 443.898,A -85,B 0,C 180,E1 -19297.511,E2 -19297.511} C_VEL
LIN {X 0,Y 266.337,Z 454.76,A -85,B 0,C 180,E1 -19300.775,E2 -19300.775} C_VEL
LIN {X 0,Y 269.12,Z 464.093,A -85,B 0,C 180,E1 -19303.275,E2 -19303.275} C_VEL
LIN {X 0,Y 271.111,Z 470.916,A -85,B 0,C 180,E1 -19304.873,E2 -19304.873} C_VEL
LIN {X 0,Y 275.569,Z 480.255,A -85,B 0,C 180,E1 -19306.127,E2 -19306.127} C_VEL
LIN {X 0,Y 279.503,Z 511.683,A -85,B 0,C 180,E1 -19307.967,E2 -19307.967} C_VEL
LIN {X 0,Y 280.8,Z 524.254,A -85,B 0,C 180,E1 -19308.626,E2 -19308.626} C_VEL
LIN {X 0,Y 275.532,Z 629.79,A -85,B 0,C 180,E1 -19311.21,E2 -19311.21} C_VEL
LIN {X 0,Y 274.283,Z 647.7,A -85,B 0,C 180,E1 -19311.763,E2 -19311.763} C_VEL
LIN {X 0,Y 272.56,Z 662.359,A -85,B 0,C 180,E1 -19312.474,E2 -19312.474} C_VEL
LIN {X 0,Y 270.28,Z 676.231,A -85,B 0,C 180,E1 -19313.389,E2 -19313.389} C_VEL
LIN {X 0,Y 267.431,Z 690.833,A -85,B 0,C 180,E1 -19314.683,E2 -19314.683} C_VEL
LIN {X 0,Y 264.183,Z 704.778,A -85,B 0,C 180,E1 -19316.27,E2 -19316.27} C_VEL
LIN {X 0,Y 260.666,Z 717.447,A -85,B 0,C 180,E1 -19318.057,E2 -19318.057} C_VEL
LIN {X 0,Y 257.174,Z 729.054,A -85,B 0,C 180,E1 -19320.087,E2 -19320.087} C_VEL
LIN {X 0,Y 253.642,Z 740.082,A -85,B 0,C 180,E1 -19322.458,E2 -19322.458} C_VEL
LIN {X 0,Y 250.864,Z 748.727,A -85,B 0,C 180,E1 -19324.711,E2 -19324.711} C_VEL
LIN {X 0,Y 247.682,Z 757.574,A -85,B 0,C 180,E1 -19327.479,E2 -19327.479} C_VEL
LIN {X 0,Y 244.856,Z 765.847,A -85,B 0,C 180,E1 -19330.729,E2 -19330.729} C_VEL
LIN {X 0,Y 242.756,Z 772.487,A -85,B 0,C 180,E1 -19334.039,E2 -19334.039} C_VEL
LIN {X 0,Y 241.184,Z 777.68,A -85,B 0,C 180,E1 -19337.379,E2 -19337.379} C_VEL
LIN {X 0,Y 240.472,Z 780.662,A -85,B 0,C 180,E1 -19339.903,E2 -19339.903} C_VEL
LIN {X 0,Y 239.895,Z 783.595,A -85,B 0,C 180,E1 -19343.273,E2 -19343.273} C_VEL
LIN {X 0,Y 239.715,Z 785.357,A -85,B 0,C 180,E1 -19346.641,E2 -19346.641} C_VEL
LIN {X 0,Y 239.771,Z 785.967,A -85,B 0,C 180,E1 -19350.003,E2 -19350.003} C_VEL
LIN {X 0,Y 239.717,Z 785.393,A -85,B 0,C 180,E1 -19353.364,E2 -19353.364} C_VEL
LIN {X 0,Y 239.898,Z 783.679,A -85,B 0,C 180,E1 -19356.732,E2 -19356.732} C_VEL
LIN {X 0,Y 240.471,Z 780.789,A -85,B 0,C 180,E1 -19360.102,E2 -19360.102} C_VEL
LIN {X 0,Y 241.49,Z 776.655,A -85,B 0,C 180,E1 -19363.466,E2 -19363.466} C_VEL
LIN {X 0,Y 243.188,Z 771.179,A -85,B 0,C 180,E1 -19366.8,E2 -19366.8} C_VEL
LIN {X 0,Y 245.421,Z 764.208,A -85,B 0,C 180,E1 -19370.101,E2 -19370.101} C_VEL
LIN {X 0,Y 248.023,Z 756.735,A -85,B 0,C 180,E1 -19372.933,E2 -19372.933} C_VEL
LIN {X 0,Y 251.213,Z 747.73,A -85,B 0,C 180,E1 -19375.701,E2 -19375.701} C_VEL
LIN {X 0,Y 254.23,Z 738.536,A -85,B 0,C 180,E1 -19378.034,E2 -19378.034} C_VEL
LIN {X 0,Y 258.061,Z 726.693,A -85,B 0,C 180,E1 -19380.482,E2 -19380.482} C_VEL
LIN {X 0,Y 261.557,Z 714.61,A -85,B 0,C 180,E1 -19382.509,E2 -19382.509} C_VEL
LIN {X 0,Y 265.159,Z 701.441,A -85,B 0,C 180,E1 -19384.266,E2 -19384.266} C_VEL
LIN {X 0,Y 268.29,Z 687.358,A -85,B 0,C 180,E1 -19385.781,E2 -19385.781} C_VEL
LIN {X 0,Y 270.93,Z 672.998,A -85,B 0,C 180,E1 -19386.979,E2 -19386.979} C_VEL
LIN {X 0,Y 273.232,Z 658.016,A -85,B 0,C 180,E1 -19387.889,E2 -19387.889} C_VEL
LIN {X 0,Y 274.892,Z 642.314,A -85,B 0,C 180,E1 -19388.551,E2 -19388.551} C_VEL
LIN {X 0,Y 276.96,Z 604.271,A -85,B 0,C 180,E1 -19389.522,E2 -19389.522} C_VEL
LIN {X 0,Y 280.925,Z 523.562,A -85,B 0,C 180,E1 -19391.509,E2 -19391.509} C_VEL
LIN {X 0,Y 276.759,Z 488.083,A -85,B 0,C 180,E1 -19393.503,E2 -19393.503} C_VEL
LIN {X 0,Y 275.431,Z 479.869,A -85,B 0,C 180,E1 -19394.055,E2 -19394.055} C_VEL
LIN {X 0,Y 270.817,Z 470.119,A -85,B 0,C 180,E1 -19395.405,E2 -19395.405} C_VEL
LIN {X 0,Y 267.932,Z 459.936,A -85,B 0,C 180,E1 -19397.988,E2 -19397.988} C_VEL
LIN {X 0,Y 264.369,Z 448.831,A -85,B 0,C 180,E1 -19401.117,E2 -19401.117} C_VEL
LIN {X 0,Y 260.909,Z 439.479,A -85,B 0,C 180,E1 -19404.087,E2 -19404.087} C_VEL
LIN {X 0,Y 257.616,Z 431.544,A -85,B 0,C 180,E1 -19406.933,E2 -19406.933} C_VEL
LIN {X 0,Y 254.617,Z 432.444,A -85,B 0,C 180,E1 -19407.773,E2 -19407.773} C_VEL
LIN {X 0,Y 254.418,Z 433.293,A -85,B 0,C 180,E1 -19408.101,E2 -19408.101} C_VEL
LIN {X 0,Y 256.579,Z 439.332,A -85,B 0,C 180,E1 -19408.63,E2 -19408.63} C_VEL
LIN {X 0,Y 257.999,Z 443.173,A -85,B 0,C 180,E1 -19408.921,E2 -19408.921} C_VEL
LIN {X 0,Y 257.239,Z 456.327,A -85,B 0,C 180,E1 -19409.478,E2 -19409.478} C_VEL
LIN {X 0,Y 256.258,Z 462.084,A -85,B 0,C 180,E1 -19409.674,E2 -19409.674} C_VEL
LIN {X 0,Y 249.555,Z 480.676,A -85,B 0,C 180,E1 -19410.096,E2 -19410.096} C_VEL
LIN {X 0,Y 248.522,Z 486.431,A -85,B 0,C 180,E1 -19410.304,E2 -19410.304} C_VEL
LIN {X 0,Y 245.41,Z 543.661,A -85,B 0,C 180,E1 -19412.901,E2 -19412.901} C_VEL
LIN {X 0,Y 244.688,Z 559.707,A -85,B 0,C 180,E1 -19413.851,E2 -19413.851} C_VEL
LIN {X 0,Y 243.59,Z 574.782,A -85,B 0,C 180,E1 -19415.042,E2 -19415.042} C_VEL
LIN {X 0,Y 242.403,Z 589.196,A -85,B 0,C 180,E1 -19416.506,E2 -19416.506} C_VEL
LIN {X 0,Y 240.985,Z 604.095,A -85,B 0,C 180,E1 -19418.396,E2 -19418.396} C_VEL
LIN {X 0,Y 239.724,Z 616.49,A -85,B 0,C 180,E1 -19420.323,E2 -19420.323} C_VEL
LIN {X 0,Y 238.388,Z 628.911,A -85,B 0,C 180,E1 -19422.632,E2 -19422.632} C_VEL
LIN {X 0,Y 237.146,Z 641.176,A -85,B 0,C 180,E1 -19425.41,E2 -19425.41} C_VEL
LIN {X 0,Y 236.335,Z 650.658,A -85,B 0,C 180,E1 -19427.985,E2 -19427.985} C_VEL
LIN {X 0,Y 235.667,Z 659.912,A -85,B 0,C 180,E1 -19430.992,E2 -19430.992} C_VEL
LIN {X 0,Y 235.128,Z 667.474,A -85,B 0,C 180,E1 -19433.995,E2 -19433.995} C_VEL
LIN {X 0,Y 235.073,Z 672.793,A -85,B 0,C 180,E1 -19436.572,E2 -19436.572} C_VEL
LIN {X 0,Y 235.32,Z 677.231,A -85,B 0,C 180,E1 -19439.144,E2 -19439.144} C_VEL
LIN {X 0,Y 235.906,Z 680.777,A -85,B 0,C 180,E1 -19441.707,E2 -19441.707} C_VEL
LIN {X 0,Y 237.124,Z 684.246,A -85,B 0,C 180,E1 -19445.101,E2 -19445.101} C_VEL
LIN {X 0,Y 238.797,Z 686.371,A -85,B 0,C 180,E1 -19448.462,E2 -19448.462} C_VEL
LIN {X 0,Y 241.204,Z 687.14,A -85,B 0,C 180,E1 -19451.768,E2 -19451.768} C_VEL
LIN {X 0,Y 244.209,Z 686.617,A -85,B 0,C 180,E1 -19455.011,E2 -19455.011} C_VEL
LIN {X 0,Y 248.034,Z 684.758,A -85,B 0,C 180,E1 -19458.161,E2 -19458.161} C_VEL
LIN {X 0,Y 252.43,Z 681.604,A -85,B 0,C 180,E1 -19461.219,E2 -19461.219} C_VEL
LIN {X 0,Y 257.539,Z 677.069,A -85,B 0,C 180,E1 -19464.163,E2 -19464.163} C_VEL
LIN {X 0,Y 263.228,Z 671.131,A -85,B 0,C 180,E1 -19466.993,E2 -19466.993} C_VEL
LIN {X 0,Y 269.613,Z 663.62,A -85,B 0,C 180,E1 -19469.688,E2 -19469.688} C_VEL
LIN {X 0,Y 275.706,Z 655.623,A -85,B 0,C 180,E1 -19471.933,E2 -19471.933} C_VEL
LIN {X 0,Y 283.125,Z 644.646,A -85,B 0,C 180,E1 -19474.383,E2 -19474.383} C_VEL
LIN {X 0,Y 290.173,Z 633.048,A -85,B 0,C 180,E1 -19476.398,E2 -19476.398} C_VEL
LIN {X 0,Y 296.518,Z 621.302,A -85,B 0,C 180,E1 -19478.042,E2 -19478.042} C_VEL
LIN {X 0,Y 303.233,Z 607.046,A -85,B 0,C 180,E1 -19479.595,E2 -19479.595} C_VEL
LIN {X 0,Y 308.351,Z 594.417,A -85,B 0,C 180,E1 -19480.725,E2 -19480.725} C_VEL
LIN {X 0,Y 313.352,Z 579.607,A -85,B 0,C 180,E1 -19481.747,E2 -19481.747} C_VEL
LIN {X 0,Y 318.468,Z 561.427,A -85,B 0,C 180,E1 -19482.733,E2 -19482.733} C_VEL
LIN {X 0,Y 317.954,Z 563.381,A -85,B 0,C 180,E1 -19482.846,E2 -19482.846} C_VEL
LIN {X 0,Y 310.793,Z 589.309,A -85,B 0,C 180,E1 -19483.878,E2 -19483.878} C_VEL
LIN {X 0,Y 305.728,Z 604.192,A -85,B 0,C 180,E1 -19484.549,E2 -19484.549} C_VEL
LIN {X 0,Y 299.288,Z 620.297,A -85,B 0,C 180,E1 -19485.447,E2 -19485.447} C_VEL
LIN {X 0,Y 291.804,Z 636.534,A -85,B 0,C 180,E1 -19486.626,E2 -19486.626} C_VEL
LIN {X 0,Y 283.352,Z 652.812,A -85,B 0,C 180,E1 -19488.148,E2 -19488.148} C_VEL
LIN {X 0,Y 276.482,Z 664.873,A -85,B 0,C 180,E1 -19489.592,E2 -19489.592} C_VEL
LIN {X 0,Y 268.626,Z 677.939,A -85,B 0,C 180,E1 -19491.582,E2 -19491.582} C_VEL
LIN {X 0,Y 261.666,Z 689.205,A -85,B 0,C 180,E1 -19493.724,E2 -19493.724} C_VEL
LIN {X 0,Y 258.202,Z 703.624,A -85,B 0,C 180,E1 -19495.373,E2 -19495.373} C_VEL
LIN {X 0,Y 254.622,Z 716.403,A -85,B 0,C 180,E1 -19497.199,E2 -19497.199} C_VEL
LIN {X 0,Y 250.985,Z 728.093,A -85,B 0,C 180,E1 -19499.265,E2 -19499.265} C_VEL
LIN {X 0,Y 247.404,Z 738.746,A -85,B 0,C 180,E1 -19501.572,E2 -19501.572} C_VEL
LIN {X 0,Y 244.365,Z 747.848,A -85,B 0,C 180,E1 -19503.983,E2 -19503.983} C_VEL
LIN {X 0,Y 241.075,Z 756.72,A -85,B 0,C 180,E1 -19506.821,E2 -19506.821} C_VEL
LIN {X 0,Y 238.082,Z 765.006,A -85,B 0,C 180,E1 -19510.153,E2 -19510.153} C_VEL
LIN {X 0,Y 235.826,Z 771.639,A -85,B 0,C 180,E1 -19513.551,E2 -19513.551} C_VEL
LIN {X 0,Y 234.232,Z 776.822,A -85,B 0,C 180,E1 -19516.993,E2 -19516.993} C_VEL
LIN {X 0,Y 233.519,Z 779.804,A -85,B 0,C 180,E1 -19519.594,E2 -19519.594} C_VEL
LIN {X 0,Y 232.916,Z 782.722,A -85,B 0,C 180,E1 -19523.065,E2 -19523.065} C_VEL
LIN {X 0,Y 232.714,Z 784.457,A -85,B 0,C 180,E1 -19526.535,E2 -19526.535} C_VEL
LIN {X 0,Y 232.778,Z 785.046,A -85,B 0,C 180,E1 -19529.997,E2 -19529.997} C_VEL
LIN {X 0,Y 232.708,Z 784.446,A -85,B 0,C 180,E1 -19533.46,E2 -19533.46} C_VEL
LIN {X 0,Y 232.91,Z 782.696,A -85,B 0,C 180,E1 -19536.93,E2 -19536.93} C_VEL
LIN {X 0,Y 233.481,Z 779.769,A -85,B 0,C 180,E1 -19540.402,E2 -19540.402} C_VEL
LIN {X 0,Y 234.576,Z 775.594,A -85,B 0,C 180,E1 -19543.865,E2 -19543.865} C_VEL
LIN {X 0,Y 236.325,Z 770.056,A -85,B 0,C 180,E1 -19547.298,E2 -19547.298} C_VEL
LIN {X 0,Y 238.716,Z 763.005,A -85,B 0,C 180,E1 -19550.686,E2 -19550.686} C_VEL
LIN {X 0,Y 241.452,Z 755.447,A -85,B 0,C 180,E1 -19553.589,E2 -19553.589} C_VEL
LIN {X 0,Y 244.787,Z 746.335,A -85,B 0,C 180,E1 -19556.421,E2 -19556.421} C_VEL
LIN {X 0,Y 247.396,Z 738.492,A -85,B 0,C 180,E1 -19558.459,E2 -19558.459} C_VEL
LIN {X 0,Y 250.935,Z 727.942,A -85,B 0,C 180,E1 -19560.736,E2 -19560.736} C_VEL
LIN {X 0,Y 254.578,Z 716.224,A -85,B 0,C 180,E1 -19562.801,E2 -19562.801} C_VEL
LIN {X 0,Y 258.112,Z 703.397,A -85,B 0,C 180,E1 -19564.635,E2 -19564.635} C_VEL
LIN {X 0,Y 261.52,Z 689.214,A -85,B 0,C 180,E1 -19566.24,E2 -19566.24} C_VEL
LIN {X 0,Y 264.256,Z 675.359,A -85,B 0,C 180,E1 -19567.468,E2 -19567.468} C_VEL
LIN {X 0,Y 266.657,Z 660.532,A -85,B 0,C 180,E1 -19568.447,E2 -19568.447} C_VEL
LIN {X 0,Y 268.473,Z 645.073,A -85,B 0,C 180,E1 -19569.16,E2 -19569.16} C_VEL
LIN {X 0,Y 269.755,Z 625.487,A -85,B 0,C 180,E1 -19569.723,E2 -19569.723} C_VEL
LIN {X 0,Y 274.003,Z 542.271,A -85,B 0,C 180,E1 -19571.789,E2 -19571.789} C_VEL
LIN {X 0,Y 275.089,Z 518.963,A -85,B 0,C 180,E1 -19572.388,E2 -19572.388} C_VEL
LIN {X 0,Y 272.486,Z 488.527,A -85,B 0,C 180,E1 -19573.972,E2 -19573.972} C_VEL
LIN {X 0,Y 271.3,Z 476.46,A -85,B 0,C 180,E1 -19574.653,E2 -19574.653} C_VEL
LIN {X 0,Y 267.629,Z 467.137,A -85,B 0,C 180,E1 -19575.829,E2 -19575.829} C_VEL
LIN {X 0,Y 262.64,Z 447.404,A -85,B 0,C 180,E1 -19579.541,E2 -19579.541} C_VEL
LIN {X 0,Y 262.132,Z 445.406,A -85,B 0,C 180,E1 -19579.95,E2 -19579.95} C_VEL
LIN {X 0,Y 257.78,Z 437.814,A -85,B 0,C 180,E1 -19582.241,E2 -19582.241} C_VEL
LIN {X 0,Y 253.19,Z 429.928,A -85,B 0,C 180,E1 -19584.942,E2 -19584.942} C_VEL
LIN {X 0,Y 248.247,Z 422.132,A -85,B 0,C 180,E1 -19588.131,E2 -19588.131} C_VEL
LIN {X 0,Y 246.692,Z 420.183,A -85,B 0,C 180,E1 -19589.15,E2 -19589.15} C_VEL
LIN {X 0,Y 244.596,Z 416.788,A -85,B 0,C 180,E1 -19590.761,E2 -19590.761} C_VEL
LIN {X 0,Y 242.522,Z 413.868,A -85,B 0,C 180,E1 -19592.377,E2 -19592.377} C_VEL
LIN {X 0,Y 241.695,Z 412.118,A -85,B 0,C 180,E1 -19593.211,E2 -19593.211} C_VEL
LIN {X 0,Y 239.754,Z 409.996,A -85,B 0,C 180,E1 -19594.847,E2 -19594.847} C_VEL
LIN {X 0,Y 238.401,Z 407.181,A -85,B 0,C 180,E1 -19596.456,E2 -19596.456} C_VEL
LIN {X 0,Y 235.822,Z 404.469,A -85,B 0,C 180,E1 -19599.046,E2 -19599.046} C_VEL
LIN {X 0,Y 234.985,Z 402.179,A -85,B 0,C 180,E1 -19600.793,E2 -19600.793} C_VEL
LIN {X 0,Y 234.982,Z 401.853,A -85,B 0,C 180,E1 -19601.697,E2 -19601.697} C_VEL
LIN {X 0,Y 235.045,Z 401.809,A -85,B 0,C 180,E1 -19606.161,E2 -19606.161} C_VEL
LIN {X 0,Y 235.275,Z 401.774,A -85,B 0,C 180,E1 -19610.297,E2 -19610.297} C_VEL
LIN {X 0,Y 235.333,Z 401.795,A -85,B 0,C 180,E1 -19613.139,E2 -19613.139} C_VEL
LIN {X 0,Y 235.562,Z 401.764,A -85,B 0,C 180,E1 -19618.291,E2 -19618.291} C_VEL
LIN {X 0,Y 235.566,Z 401.739,A -85,B 0,C 180,E1 -19621.71,E2 -19621.71} C_VEL
LIN {X 0,Y 235.342,Z 401.766,A -85,B 0,C 180,E1 -19626.861,E2 -19626.861} C_VEL
LIN {X 0,Y 235.172,Z 401.796,A -85,B 0,C 180,E1 -19630.33,E2 -19630.33} C_VEL
LIN {X 0,Y 235.118,Z 402.113,A -85,B 0,C 180,E1 -19632.955,E2 -19632.955} C_VEL
LIN {X 0,Y 236.359,Z 405.117,A -85,B 0,C 180,E1 -19635.522,E2 -19635.522} C_VEL
LIN {X 0,Y 237.847,Z 406.692,A -85,B 0,C 180,E1 -19637.187,E2 -19637.187} C_VEL
LIN {X 0,Y 239.676,Z 410.459,A -85,B 0,C 180,E1 -19639.707,E2 -19639.707} C_VEL
LIN {X 0,Y 240.794,Z 412.085,A -85,B 0,C 180,E1 -19640.946,E2 -19640.946} C_VEL
LIN {X 0,Y 245.037,Z 419.94,A -85,B 0,C 180,E1 -19645.482,E2 -19645.482} C_VEL
LIN {X 0,Y 249.225,Z 428.421,A -85,B 0,C 180,E1 -19649.57,E2 -19649.57} C_VEL
LIN {X 0,Y 253.187,Z 437.374,A -85,B 0,C 180,E1 -19653.245,E2 -19653.245} C_VEL
LIN {X 0,Y 257.252,Z 447.923,A -85,B 0,C 180,E1 -19656.944,E2 -19656.944} C_VEL
LIN {X 0,Y 260.61,Z 457.7,A -85,B 0,C 180,E1 -19659.957,E2 -19659.957} C_VEL
LIN {X 0,Y 263.408,Z 467.102,A -85,B 0,C 180,E1 -19662.553,E2 -19662.553} C_VEL
LIN {X 0,Y 264.576,Z 470.919,A -85,B 0,C 180,E1 -19663.44,E2 -19663.44} C_VEL
LIN {X 0,Y 270.692,Z 483.544,A -85,B 0,C 180,E1 -19665.25,E2 -19665.25} C_VEL
LIN {X 0,Y 274.83,Z 518.388,A -85,B 0,C 180,E1 -19667.32,E2 -19667.32} C_VEL
LIN {X 0,Y 275.44,Z 525.389,A -85,B 0,C 180,E1 -19667.68,E2 -19667.68} C_VEL
LIN {X 0,Y 270.046,Z 629.688,A -85,B 0,C 180,E1 -19670.268,E2 -19670.268} C_VEL
LIN {X 0,Y 268.753,Z 647.64,A -85,B 0,C 180,E1 -19670.828,E2 -19670.828} C_VEL
LIN {X 0,Y 266.978,Z 662.317,A -85,B 0,C 180,E1 -19671.548,E2 -19671.548} C_VEL
LIN {X 0,Y 264.607,Z 676.199,A -85,B 0,C 180,E1 -19672.47,E2 -19672.47} C_VEL
LIN {X 0,Y 261.657,Z 690.807,A -85,B 0,C 180,E1 -19673.782,E2 -19673.782} C_VEL
LIN {X 0,Y 258.292,Z 704.755,A -85,B 0,C 180,E1 -19675.393,E2 -19675.393} C_VEL
LIN {X 0,Y 254.64,Z 717.427,A -85,B 0,C 180,E1 -19677.208,E2 -19677.208} C_VEL
LIN {X 0,Y 251.023,Z 729.036,A -85,B 0,C 180,E1 -19679.276,E2 -19679.276} C_VEL
LIN {X 0,Y 247.094,Z 740.718,A -85,B 0,C 180,E1 -19681.851,E2 -19681.851} C_VEL
LIN {X 0,Y 243.892,Z 750.048,A -85,B 0,C 180,E1 -19684.393,E2 -19684.393} C_VEL
LIN {X 0,Y 240.676,Z 758.662,A -85,B 0,C 180,E1 -19687.24,E2 -19687.24} C_VEL
LIN {X 0,Y 238.104,Z 765.832,A -85,B 0,C 180,E1 -19690.16,E2 -19690.16} C_VEL
LIN {X 0,Y 235.872,Z 772.473,A -85,B 0,C 180,E1 -19693.56,E2 -19693.56} C_VEL
LIN {X 0,Y 234.216,Z 777.667,A -85,B 0,C 180,E1 -19696.997,E2 -19696.997} C_VEL
LIN {X 0,Y 233.449,Z 780.648,A -85,B 0,C 180,E1 -19699.596,E2 -19699.596} C_VEL
LIN {X 0,Y 232.816,Z 783.582,A -85,B 0,C 180,E1 -19703.068,E2 -19703.068} C_VEL
LIN {X 0,Y 232.627,Z 785.343,A -85,B 0,C 180,E1 -19706.539,E2 -19706.539} C_VEL
LIN {X 0,Y 232.687,Z 785.953,A -85,B 0,C 180,E1 -19710.003,E2 -19710.003} C_VEL
LIN {X 0,Y 232.628,Z 785.379,A -85,B 0,C 180,E1 -19713.467,E2 -19713.467} C_VEL
LIN {X 0,Y 232.819,Z 783.665,A -85,B 0,C 180,E1 -19716.938,E2 -19716.938} C_VEL
LIN {X 0,Y 233.447,Z 780.774,A -85,B 0,C 180,E1 -19720.409,E2 -19720.409} C_VEL
LIN {X 0,Y 234.56,Z 776.639,A -85,B 0,C 180,E1 -19723.871,E2 -19723.871} C_VEL
LIN {X 0,Y 236.349,Z 771.163,A -85,B 0,C 180,E1 -19727.301,E2 -19727.301} C_VEL
LIN {X 0,Y 238.701,Z 764.19,A -85,B 0,C 180,E1 -19730.693,E2 -19730.693} C_VEL
LIN {X 0,Y 241.417,Z 756.716,A -85,B 0,C 180,E1 -19733.598,E2 -19733.598} C_VEL
LIN {X 0,Y 244.785,Z 747.709,A -85,B 0,C 180,E1 -19736.427,E2 -19736.427} C_VEL
LIN {X 0,Y 247.929,Z 738.514,A -85,B 0,C 180,E1 -19738.812,E2 -19738.812} C_VEL
LIN {X 0,Y 251.932,Z 726.668,A -85,B 0,C 180,E1 -19741.306,E2 -19741.306} C_VEL
LIN {X 0,Y 255.578,Z 714.582,A -85,B 0,C 180,E1 -19743.367,E2 -19743.367} C_VEL
LIN {X 0,Y 259.272,Z 701.584,A -85,B 0,C 180,E1 -19745.128,E2 -19745.128} C_VEL
LIN {X 0,Y 262.467,Z 687.689,A -85,B 0,C 180,E1 -19746.654,E2 -19746.654} C_VEL
LIN {X 0,Y 265.299,Z 672.946,A -85,B 0,C 180,E1 -19747.9,E2 -19747.9} C_VEL
LIN {X 0,Y 267.65,Z 657.943,A -85,B 0,C 180,E1 -19748.825,E2 -19748.825} C_VEL
LIN {X 0,Y 269.365,Z 642.199,A -85,B 0,C 180,E1 -19749.494,E2 -19749.494} C_VEL
LIN {X 0,Y 271.794,Z 598.508,A -85,B 0,C 180,E1 -19750.618,E2 -19750.618} C_VEL
LIN {X 0,Y 275.593,Z 525.242,A -85,B 0,C 180,E1 -19752.434,E2 -19752.434} C_VEL
LIN {X 0,Y 272.325,Z 495.57,A -85,B 0,C 180,E1 -19754.12,E2 -19754.12} C_VEL
LIN {X 0,Y 270.687,Z 483.371,A -85,B 0,C 180,E1 -19754.901,E2 -19754.901} C_VEL
LIN {X 0,Y 264.249,Z 469.845,A -85,B 0,C 180,E1 -19756.89,E2 -19756.89} C_VEL
LIN {X 0,Y 260.198,Z 456.341,A -85,B 0,C 180,E1 -19760.599,E2 -19760.599} C_VEL
LIN {X 0,Y 256.793,Z 446.495,A -85,B 0,C 180,E1 -19763.692,E2 -19763.692} C_VEL
LIN {X 0,Y 253.833,Z 438.863,A -85,B 0,C 180,E1 -19766.375,E2 -19766.375} C_VEL
LIN {X 0,Y 252.044,Z 438.457,A -85,B 0,C 180,E1 -19767.061,E2 -19767.061} C_VEL
LIN {X 0,Y 250.005,Z 439.18,A -85,B 0,C 180,E1 -19767.597,E2 -19767.597} C_VEL
LIN {X 0,Y 249.54,Z 439.719,A -85,B 0,C 180,E1 -19767.94,E2 -19767.94} C_VEL
LIN {X 0,Y 249.664,Z 440.474,A -85,B 0,C 180,E1 -19768.104,E2 -19768.104} C_VEL
LIN {X 0,Y 251.237,Z 445.121,A -85,B 0,C 180,E1 -19768.496,E2 -19768.496} C_VEL
LIN {X 0,Y 248.522,Z 486.431,A -85,B 0,C 180,E1 -19770.304,E2 -19770.304} C_VEL
LIN {X 0,Y 247.479,Z 492.188,A -85,B 0,C 180,E1 -19770.513,E2 -19770.513} C_VEL
LIN {X 0,Y 240.769,Z 510.766,A -85,B 0,C 180,E1 -19771,E2 -19771} C_VEL
LIN {X 0,Y 239.831,Z 516.518,A -85,B 0,C 180,E1 -19771.229,E2 -19771.229} C_VEL
LIN {X 0,Y 238.049,Z 552.443,A -85,B 0,C 180,E1 -19773.004,E2 -19773.004} C_VEL
LIN {X 0,Y 237.228,Z 567.608,A -85,B 0,C 180,E1 -19774.089,E2 -19774.089} C_VEL
LIN {X 0,Y 235.951,Z 582.596,A -85,B 0,C 180,E1 -19775.472,E2 -19775.472} C_VEL
LIN {X 0,Y 234.781,Z 596.497,A -85,B 0,C 180,E1 -19777.098,E2 -19777.098} C_VEL
LIN {X 0,Y 233.235,Z 610.662,A -85,B 0,C 180,E1 -19779.128,E2 -19779.128} C_VEL
LIN {X 0,Y 231.944,Z 623.964,A -85,B 0,C 180,E1 -19781.448,E2 -19781.448} C_VEL
LIN {X 0,Y 230.518,Z 636.403,A -85,B 0,C 180,E1 -19784.074,E2 -19784.074} C_VEL
LIN {X 0,Y 229.588,Z 646.837,A -85,B 0,C 180,E1 -19786.727,E2 -19786.727} C_VEL
LIN {X 0,Y 228.862,Z 655.617,A -85,B 0,C 180,E1 -19789.382,E2 -19789.382} C_VEL
LIN {X 0,Y 228.343,Z 663.036,A -85,B 0,C 180,E1 -19792.039,E2 -19792.039} C_VEL
LIN {X 0,Y 228.001,Z 669.324,A -85,B 0,C 180,E1 -19794.694,E2 -19794.694} C_VEL
LIN {X 0,Y 228.151,Z 676.109,A -85,B 0,C 180,E1 -19798.235,E2 -19798.235} C_VEL
LIN {X 0,Y 228.523,Z 680.162,A -85,B 0,C 180,E1 -19800.881,E2 -19800.881} C_VEL
LIN {X 0,Y 229.38,Z 683.325,A -85,B 0,C 180,E1 -19803.513,E2 -19803.513} C_VEL
LIN {X 0,Y 230.925,Z 686.393,A -85,B 0,C 180,E1 -19806.992,E2 -19806.992} C_VEL
LIN {X 0,Y 232.965,Z 688.137,A -85,B 0,C 180,E1 -19810.428,E2 -19810.428} C_VEL
LIN {X 0,Y 235.866,Z 688.544,A -85,B 0,C 180,E1 -19813.79,E2 -19813.79} C_VEL
LIN {X 0,Y 239.48,Z 687.665,A -85,B 0,C 180,E1 -19817.066,E2 -19817.066} C_VEL
LIN {X 0,Y 243.797,Z 685.514,A -85,B 0,C 180,E1 -19820.238,E2 -19820.238} C_VEL
LIN {X 0,Y 248.751,Z 682.081,A -85,B 0,C 180,E1 -19823.3,E2 -19823.3} C_VEL
LIN {X 0,Y 254.472,Z 677.257,A -85,B 0,C 180,E1 -19826.224,E2 -19826.224} C_VEL
LIN {X 0,Y 260.764,Z 671.037,A -85,B 0,C 180,E1 -19829.021,E2 -19829.021} C_VEL
LIN {X 0,Y 267.757,Z 663.191,A -85,B 0,C 180,E1 -19831.665,E2 -19831.665} C_VEL
LIN {X 0,Y 275.304,Z 653.698,A -85,B 0,C 180,E1 -19834.168,E2 -19834.168} C_VEL
LIN {X 0,Y 282.378,Z 643.75,A -85,B 0,C 180,E1 -19836.235,E2 -19836.235} C_VEL
LIN {X 0,Y 289.89,Z 631.882,A -85,B 0,C 180,E1 -19838.186,E2 -19838.186} C_VEL
LIN {X 0,Y 296.174,Z 620.789,A -85,B 0,C 180,E1 -19839.622,E2 -19839.622} C_VEL
LIN {X 0,Y 302.345,Z 608.445,A -85,B 0,C 180,E1 -19840.936,E2 -19840.936} C_VEL
LIN {X 0,Y 308.059,Z 595.153,A -85,B 0,C 180,E1 -19842.079,E2 -19842.079} C_VEL
LIN {X 0,Y 309.425,Z 591.508,A -85,B 0,C 180,E1 -19842.338,E2 -19842.338} C_VEL
LIN {X 0,Y 309.689,Z 590.984,A -85,B 0,C 180,E1 -19842.617,E2 -19842.617} C_VEL
LIN {X 0,Y 303.373,Z 607.703,A -85,B 0,C 180,E1 -19843.376,E2 -19843.376} C_VEL
LIN {X 0,Y 296.757,Z 622.707,A -85,B 0,C 180,E1 -19844.24,E2 -19844.24} C_VEL
LIN {X 0,Y 288.975,Z 638.262,A -85,B 0,C 180,E1 -19845.39,E2 -19845.39} C_VEL
LIN {X 0,Y 279.997,Z 654.141,A -85,B 0,C 180,E1 -19846.91,E2 -19846.91} C_VEL
LIN {X 0,Y 272.016,Z 667.066,A -85,B 0,C 180,E1 -19848.515,E2 -19848.515} C_VEL
LIN {X 0,Y 263.282,Z 680.328,A -85,B 0,C 180,E1 -19850.653,E2 -19850.653} C_VEL
LIN {X 0,Y 255.352,Z 692.14,A -85,B 0,C 180,E1 -19853.089,E2 -19853.089} C_VEL
LIN {X 0,Y 251.624,Z 706.476,A -85,B 0,C 180,E1 -19854.823,E2 -19854.823} C_VEL
LIN {X 0,Y 247.954,Z 718.756,A -85,B 0,C 180,E1 -19856.688,E2 -19856.688} C_VEL
LIN {X 0,Y 244.2,Z 730.054,A -85,B 0,C 180,E1 -19858.797,E2 -19858.797} C_VEL
LIN {X 0,Y 240.364,Z 740.936,A -85,B 0,C 180,E1 -19861.302,E2 -19861.302} C_VEL
LIN {X 0,Y 236.899,Z 750.558,A -85,B 0,C 180,E1 -19864.048,E2 -19864.048} C_VEL
LIN {X 0,Y 233.664,Z 758.958,A -85,B 0,C 180,E1 -19866.98,E2 -19866.98} C_VEL
LIN {X 0,Y 230.677,Z 766.821,A -85,B 0,C 180,E1 -19870.417,E2 -19870.417} C_VEL
LIN {X 0,Y 228.527,Z 773.07,A -85,B 0,C 180,E1 -19873.929,E2 -19873.929} C_VEL
LIN {X 0,Y 226.957,Z 777.897,A -85,B 0,C 180,E1 -19877.478,E2 -19877.478} C_VEL
LIN {X 0,Y 226.125,Z 781.429,A -85,B 0,C 180,E1 -19881.057,E2 -19881.057} C_VEL
LIN {X 0,Y 225.692,Z 783.99,A -85,B 0,C 180,E1 -19885.184,E2 -19885.184} C_VEL
LIN {X 0,Y 225.646,Z 784.909,A -85,B 0,C 180,E1 -19888.212,E2 -19888.212} C_VEL
LIN {X 0,Y 225.693,Z 785.059,A -85,B 0,C 180,E1 -19889.997,E2 -19889.997} C_VEL
LIN {X 0,Y 225.619,Z 784.459,A -85,B 0,C 180,E1 -19893.569,E2 -19893.569} C_VEL
LIN {X 0,Y 225.833,Z 782.71,A -85,B 0,C 180,E1 -19897.148,E2 -19897.148} C_VEL
LIN {X 0,Y 226.468,Z 779.783,A -85,B 0,C 180,E1 -19900.728,E2 -19900.728} C_VEL
LIN {X 0,Y 227.661,Z 775.608,A -85,B 0,C 180,E1 -19904.295,E2 -19904.295} C_VEL
LIN {X 0,Y 229.496,Z 770.07,A -85,B 0,C 180,E1 -19907.829,E2 -19907.829} C_VEL
LIN {X 0,Y 232.049,Z 763.02,A -85,B 0,C 180,E1 -19911.308,E2 -19911.308} C_VEL
LIN {X 0,Y 234.882,Z 755.463,A -85,B 0,C 180,E1 -19914.291,E2 -19914.291} C_VEL
LIN {X 0,Y 238.386,Z 746.351,A -85,B 0,C 180,E1 -19917.188,E2 -19917.188} C_VEL
LIN {X 0,Y 241.068,Z 738.683,A -85,B 0,C 180,E1 -19919.226,E2 -19919.226} C_VEL
LIN {X 0,Y 244.829,Z 727.96,A -85,B 0,C 180,E1 -19921.589,E2 -19921.589} C_VEL
LIN {X 0,Y 248.626,Z 716.245,A -85,B 0,C 180,E1 -19923.69,E2 -19923.69} C_VEL
LIN {X 0,Y 252.293,Z 703.42,A -85,B 0,C 180,E1 -19925.553,E2 -19925.553} C_VEL
LIN {X 0,Y 255.815,Z 689.241,A -85,B 0,C 180,E1 -19927.182,E2 -19927.182} C_VEL
LIN {X 0,Y 258.656,Z 675.389,A -85,B 0,C 180,E1 -19928.425,E2 -19928.425} C_VEL
LIN {X 0,Y 261.151,Z 660.575,A -85,B 0,C 180,E1 -19929.412,E2 -19929.412} C_VEL
LIN {X 0,Y 263.022,Z 645.135,A -85,B 0,C 180,E1 -19930.134,E2 -19930.134} C_VEL
LIN {X 0,Y 264.334,Z 625.592,A -85,B 0,C 180,E1 -19930.706,E2 -19930.706} C_VEL
LIN {X 0,Y 268.749,Z 542.376,A -85,B 0,C 180,E1 -19932.798,E2 -19932.798} C_VEL
LIN {X 0,Y 269.85,Z 519.803,A -85,B 0,C 180,E1 -19933.385,E2 -19933.385} C_VEL
LIN {X 0,Y 267.282,Z 488.169,A -85,B 0,C 180,E1 -19935.076,E2 -19935.076} C_VEL
LIN {X 0,Y 266.366,Z 479.217,A -85,B 0,C 180,E1 -19935.611,E2 -19935.611} C_VEL
LIN {X 0,Y 261.656,Z 467.412,A -85,B 0,C 180,E1 -19937.165,E2 -19937.165} C_VEL
LIN {X 0,Y 257.949,Z 451.895,A -85,B 0,C 180,E1 -19940.187,E2 -19940.187} C_VEL
LIN {X 0,Y 257.456,Z 449.931,A -85,B 0,C 180,E1 -19940.604,E2 -19940.604} C_VEL
LIN {X 0,Y 252.081,Z 440.308,A -85,B 0,C 180,E1 -19943.669,E2 -19943.669} C_VEL
LIN {X 0,Y 247.653,Z 432.944,A -85,B 0,C 180,E1 -19946.401,E2 -19946.401} C_VEL
LIN {X 0,Y 244.137,Z 427.453,A -85,B 0,C 180,E1 -19948.791,E2 -19948.791} C_VEL
LIN {X 0,Y 240.912,Z 422.569,A -85,B 0,C 180,E1 -19951.226,E2 -19951.226} C_VEL
LIN {X 0,Y 238.097,Z 418.015,A -85,B 0,C 180,E1 -19953.72,E2 -19953.72} C_VEL
LIN {X 0,Y 235.742,Z 414.808,A -85,B 0,C 180,E1 -19955.931,E2 -19955.931} C_VEL
LIN {X 0,Y 234.681,Z 413.051,A -85,B 0,C 180,E1 -19957.089,E2 -19957.089} C_VEL
LIN {X 0,Y 232.399,Z 410.29,A -85,B 0,C 180,E1 -19959.622,E2 -19959.622} C_VEL
LIN {X 0,Y 231.877,Z 409.012,A -85,B 0,C 180,E1 -19960.525,E2 -19960.525} C_VEL
LIN {X 0,Y 228.115,Z 403.132,A -85,B 0,C 180,E1 -19967.772,E2 -19967.772} C_VEL
LIN {X 0,Y 228.215,Z 402.66,A -85,B 0,C 180,E1 -19970.196,E2 -19970.196} C_VEL
LIN {X 0,Y 228.286,Z 402.67,A -85,B 0,C 180,E1 -19972.927,E2 -19972.927} C_VEL
LIN {X 0,Y 228.521,Z 402.639,A -85,B 0,C 180,E1 -19978.238,E2 -19978.238} C_VEL
LIN {X 0,Y 228.524,Z 402.616,A -85,B 0,C 180,E1 -19981.763,E2 -19981.763} C_VEL
LIN {X 0,Y 228.205,Z 402.933,A -85,B 0,C 180,E1 -19985.745,E2 -19985.745} C_VEL
LIN {X 0,Y 228.459,Z 403.57,A -85,B 0,C 180,E1 -19987.068,E2 -19987.068} C_VEL
LIN {X 0,Y 229.79,Z 406.441,A -85,B 0,C 180,E1 -19990.574,E2 -19990.574} C_VEL
LIN {X 0,Y 230.95,Z 407.579,A -85,B 0,C 180,E1 -19992.299,E2 -19992.299} C_VEL
LIN {X 0,Y 234.175,Z 413.376,A -85,B 0,C 180,E1 -19997.465,E2 -19997.465} C_VEL
LIN {X 0,Y 236.837,Z 418.177,A -85,B 0,C 180,E1 -20000.861,E2 -20000.861} C_VEL
LIN {X 0,Y 240.587,Z 425.244,A -85,B 0,C 180,E1 -20005.108,E2 -20005.108} C_VEL
LIN {X 0,Y 244.635,Z 433.608,A -85,B 0,C 180,E1 -20009.235,E2 -20009.235} C_VEL
LIN {X 0,Y 248.512,Z 442.657,A -85,B 0,C 180,E1 -20012.984,E2 -20012.984} C_VEL
LIN {X 0,Y 252.471,Z 453.266,A -85,B 0,C 180,E1 -20016.762,E2 -20016.762} C_VEL
LIN {X 0,Y 256.027,Z 464.246,A -85,B 0,C 180,E1 -20020.171,E2 -20020.171} C_VEL
LIN {X 0,Y 258.077,Z 470.793,A -85,B 0,C 180,E1 -20021.894,E2 -20021.894} C_VEL
LIN {X 0,Y 264.577,Z 483.999,A -85,B 0,C 180,E1 -20023.945,E2 -20023.945} C_VEL
LIN {X 0,Y 265.994,Z 487.421,A -85,B 0,C 180,E1 -20024.389,E2 -20024.389} C_VEL
LIN {X 0,Y 270.126,Z 524.542,A -85,B 0,C 180,E1 -20026.618,E2 -20026.618} C_VEL
LIN {X 0,Y 269.26,Z 544.007,A -85,B 0,C 180,E1 -20027.143,E2 -20027.143} C_VEL
LIN {X 0,Y 263.941,Z 640.53,A -85,B 0,C 180,E1 -20029.597,E2 -20029.597} C_VEL
LIN {X 0,Y 262.302,Z 656.036,A -85,B 0,C 180,E1 -20030.235,E2 -20030.235} C_VEL
LIN {X 0,Y 260.075,Z 670.316,A -85,B 0,C 180,E1 -20031.08,E2 -20031.08} C_VEL
LIN {X 0,Y 257.293,Z 684.841,A -85,B 0,C 180,E1 -20032.262,E2 -20032.262} C_VEL
LIN {X 0,Y 254.279,Z 697.862,A -85,B 0,C 180,E1 -20033.626,E2 -20033.626} C_VEL
LIN {X 0,Y 250.547,Z 711.372,A -85,B 0,C 180,E1 -20035.391,E2 -20035.391} C_VEL
LIN {X 0,Y 246.562,Z 723.995,A -85,B 0,C 180,E1 -20037.455,E2 -20037.455} C_VEL
LIN {X 0,Y 242.996,Z 734.569,A -85,B 0,C 180,E1 -20039.596,E2 -20039.596} C_VEL
LIN {X 0,Y 239.598,Z 744.358,A -85,B 0,C 180,E1 -20042.013,E2 -20042.013} C_VEL
LIN {X 0,Y 235.914,Z 753.929,A -85,B 0,C 180,E1 -20044.883,E2 -20044.883} C_VEL
LIN {X 0,Y 232.881,Z 761.9,A -85,B 0,C 180,E1 -20047.841,E2 -20047.841} C_VEL
LIN {X 0,Y 230.218,Z 769.054,A -85,B 0,C 180,E1 -20051.148,E2 -20051.148} C_VEL
LIN {X 0,Y 228.102,Z 775.228,A -85,B 0,C 180,E1 -20054.821,E2 -20054.821} C_VEL
LIN {X 0,Y 226.924,Z 778.708,A -85,B 0,C 180,E1 -20057.482,E2 -20057.482} C_VEL
LIN {X 0,Y 226.024,Z 782.251,A -85,B 0,C 180,E1 -20061.059,E2 -20061.059} C_VEL
LIN {X 0,Y 225.591,Z 784.592,A -85,B 0,C 180,E1 -20064.64,E2 -20064.64} C_VEL
LIN {X 0,Y 225.546,Z 785.782,A -85,B 0,C 180,E1 -20068.217,E2 -20068.217} C_VEL
LIN {X 0,Y 225.586,Z 785.939,A -85,B 0,C 180,E1 -20070.003,E2 -20070.003} C_VEL
LIN {X 0,Y 225.525,Z 785.365,A -85,B 0,C 180,E1 -20073.576,E2 -20073.576} C_VEL
LIN {X 0,Y 225.765,Z 783.65,A -85,B 0,C 180,E1 -20077.156,E2 -20077.156} C_VEL
LIN {X 0,Y 226.437,Z 780.759,A -85,B 0,C 180,E1 -20080.735,E2 -20080.735} C_VEL
LIN {X 0,Y 227.642,Z 776.624,A -85,B 0,C 180,E1 -20084.302,E2 -20084.302} C_VEL
LIN {X 0,Y 229.531,Z 771.146,A -85,B 0,C 180,E1 -20087.832,E2 -20087.832} C_VEL
LIN {X 0,Y 232.033,Z 764.173,A -85,B 0,C 180,E1 -20091.316,E2 -20091.316} C_VEL
LIN {X 0,Y 234.875,Z 756.697,A -85,B 0,C 180,E1 -20094.297,E2 -20094.297} C_VEL
LIN {X 0,Y 238.397,Z 747.689,A -85,B 0,C 180,E1 -20097.193,E2 -20097.193} C_VEL
LIN {X 0,Y 241.692,Z 738.492,A -85,B 0,C 180,E1 -20099.628,E2 -20099.628} C_VEL
LIN {X 0,Y 245.862,Z 726.643,A -85,B 0,C 180,E1 -20102.17,E2 -20102.17} C_VEL
LIN {X 0,Y 249.651,Z 714.553,A -85,B 0,C 180,E1 -20104.268,E2 -20104.268} C_VEL
LIN {X 0,Y 253.433,Z 701.765,A -85,B 0,C 180,E1 -20106.025,E2 -20106.025} C_VEL
LIN {X 0,Y 256.801,Z 687.649,A -85,B 0,C 180,E1 -20107.6,E2 -20107.6} C_VEL
LIN {X 0,Y 259.52,Z 674.039,A -85,B 0,C 180,E1 -20108.776,E2 -20108.776} C_VEL
LIN {X 0,Y 262.055,Z 658.689,A -85,B 0,C 180,E1 -20109.754,E2 -20109.754} C_VEL
LIN {X 0,Y 263.837,Z 643.405,A -85,B 0,C 180,E1 -20110.428,E2 -20110.428} C_VEL
LIN {X 0,Y 265.267,Z 620.878,A -85,B 0,C 180,E1 -20111.04,E2 -20111.04} C_VEL
LIN {X 0,Y 270.323,Z 525.707,A -85,B 0,C 180,E1 -20113.441,E2 -20113.441} C_VEL
LIN {X 0,Y 266.63,Z 491.809,A -85,B 0,C 180,E1 -20115.454,E2 -20115.454} C_VEL
LIN {X 0,Y 265.775,Z 486.466,A -85,B 0,C 180,E1 -20115.843,E2 -20115.843} C_VEL
LIN {X 0,Y 259.571,Z 473.609,A -85,B 0,C 180,E1 -20117.778,E2 -20117.778} C_VEL
LIN {X 0,Y 257.68,Z 469.807,A -85,B 0,C 180,E1 -20118.461,E2 -20118.461} C_VEL
LIN {X 0,Y 254.791,Z 459.995,A -85,B 0,C 180,E1 -20121.296,E2 -20121.296} C_VEL
LIN {X 0,Y 251.767,Z 451.143,A -85,B 0,C 180,E1 -20124.111,E2 -20124.111} C_VEL
LIN {X 0,Y 249.373,Z 444.759,A -85,B 0,C 180,E1 -20126.4,E2 -20126.4} C_VEL
LIN {X 0,Y 247.739,Z 445.107,A -85,B 0,C 180,E1 -20126.858,E2 -20126.858} C_VEL
LIN {X 0,Y 245.132,Z 446.015,A -85,B 0,C 180,E1 -20127.548,E2 -20127.548} C_VEL
LIN {X 0,Y 244.604,Z 446.736,A -85,B 0,C 180,E1 -20127.902,E2 -20127.902} C_VEL
LIN {X 0,Y 244.272,Z 449.535,A -85,B 0,C 180,E1 -20128.153,E2 -20128.153} C_VEL
LIN {X 0,Y 239.831,Z 516.518,A -85,B 0,C 180,E1 -20131.229,E2 -20131.229} C_VEL
LIN {X 0,Y 238.947,Z 522.262,A -85,B 0,C 180,E1 -20131.464,E2 -20131.464} C_VEL
LIN {X 0,Y 233.127,Z 538.975,A -85,B 0,C 180,E1 -20131.989,E2 -20131.989} C_VEL
LIN {X 0,Y 231.722,Z 544.652,A -85,B 0,C 180,E1 -20132.223,E2 -20132.223} C_VEL
LIN {X 0,Y 231.477,Z 546.573,A -85,B 0,C 180,E1 -20132.319,E2 -20132.319} C_VEL
LIN {X 0,Y 230.653,Z 562.511,A -85,B 0,C 180,E1 -20133.354,E2 -20133.354} C_VEL
LIN {X 0,Y 229.358,Z 578.231,A -85,B 0,C 180,E1 -20134.718,E2 -20134.718} C_VEL
LIN {X 0,Y 228.058,Z 593.117,A -85,B 0,C 180,E1 -20136.383,E2 -20136.383} C_VEL
LIN {X 0,Y 226.608,Z 607.674,A -85,B 0,C 180,E1 -20138.399,E2 -20138.399} C_VEL
LIN {X 0,Y 225.174,Z 620.879,A -85,B 0,C 180,E1 -20140.633,E2 -20140.633} C_VEL
LIN {X 0,Y 223.83,Z 633.024,A -85,B 0,C 180,E1 -20143.116,E2 -20143.116} C_VEL
LIN {X 0,Y 222.765,Z 644.108,A -85,B 0,C 180,E1 -20145.847,E2 -20145.847} C_VEL
LIN {X 0,Y 221.953,Z 653.461,A -85,B 0,C 180,E1 -20148.586,E2 -20148.586} C_VEL
LIN {X 0,Y 221.313,Z 662.627,A -85,B 0,C 180,E1 -20151.784,E2 -20151.784} C_VEL
LIN {X 0,Y 220.912,Z 669.159,A -85,B 0,C 180,E1 -20154.523,E2 -20154.523} C_VEL
LIN {X 0,Y 221.05,Z 676.269,A -85,B 0,C 180,E1 -20158.178,E2 -20158.178} C_VEL
LIN {X 0,Y 221.438,Z 680.505,A -85,B 0,C 180,E1 -20160.909,E2 -20160.909} C_VEL
LIN {X 0,Y 222.332,Z 683.965,A -85,B 0,C 180,E1 -20163.625,E2 -20163.625} C_VEL
LIN {X 0,Y 223.945,Z 687.293,A -85,B 0,C 180,E1 -20167.211,E2 -20167.211} C_VEL
LIN {X 0,Y 226.099,Z 689.323,A -85,B 0,C 180,E1 -20170.749,E2 -20170.749} C_VEL
LIN {X 0,Y 229.14,Z 690.035,A -85,B 0,C 180,E1 -20174.203,E2 -20174.203} C_VEL
LIN {X 0,Y 232.925,Z 689.475,A -85,B 0,C 180,E1 -20177.561,E2 -20177.561} C_VEL
LIN {X 0,Y 237.476,Z 687.65,A -85,B 0,C 180,E1 -20180.802,E2 -20180.802} C_VEL
LIN {X 0,Y 242.663,Z 684.584,A -85,B 0,C 180,E1 -20183.92,E2 -20183.92} C_VEL
LIN {X 0,Y 248.646,Z 680.157,A -85,B 0,C 180,E1 -20186.887,E2 -20186.887} C_VEL
LIN {X 0,Y 255.214,Z 674.407,A -85,B 0,C 180,E1 -20189.714,E2 -20189.714} C_VEL
LIN {X 0,Y 262.462,Z 667.191,A -85,B 0,C 180,E1 -20192.381,E2 -20192.381} C_VEL
LIN {X 0,Y 270.34,Z 658.331,A -85,B 0,C 180,E1 -20194.885,E2 -20194.885} C_VEL
LIN {X 0,Y 277.688,Z 649.049,A -85,B 0,C 180,E1 -20196.948,E2 -20196.948} C_VEL
LIN {X 0,Y 285.511,Z 638.077,A -85,B 0,C 180,E1 -20198.88,E2 -20198.88} C_VEL
LIN {X 0,Y 293.15,Z 626.035,A -85,B 0,C 180,E1 -20200.564,E2 -20200.564} C_VEL
LIN {X 0,Y 299.912,Z 613.804,A -85,B 0,C 180,E1 -20201.902,E2 -20201.902} C_VEL
LIN {X 0,Y 300.295,Z 613.246,A -85,B 0,C 180,E1 -20202.293,E2 -20202.293} C_VEL
LIN {X 0,Y 292.904,Z 628.187,A -85,B 0,C 180,E1 -20203.21,E2 -20203.21} C_VEL
LIN {X 0,Y 284.962,Z 642.46,A -85,B 0,C 180,E1 -20204.336,E2 -20204.336} C_VEL
LIN {X 0,Y 276.071,Z 656.814,A -85,B 0,C 180,E1 -20205.776,E2 -20205.776} C_VEL
LIN {X 0,Y 267.666,Z 669.314,A -85,B 0,C 180,E1 -20207.406,E2 -20207.406} C_VEL
LIN {X 0,Y 259.158,Z 681.181,A -85,B 0,C 180,E1 -20209.392,E2 -20209.392} C_VEL
LIN {X 0,Y 250.537,Z 692.717,A -85,B 0,C 180,E1 -20211.89,E2 -20211.89} C_VEL
LIN {X 0,Y 248.98,Z 695.096,A -85,B 0,C 180,E1 -20212.439,E2 -20212.439} C_VEL
LIN {X 0,Y 245.063,Z 709.101,A -85,B 0,C 180,E1 -20214.242,E2 -20214.242} C_VEL
LIN {X 0,Y 241.333,Z 720.969,A -85,B 0,C 180,E1 -20216.152,E2 -20216.152} C_VEL
LIN {X 0,Y 237.446,Z 731.951,A -85,B 0,C 180,E1 -20218.304,E2 -20218.304} C_VEL
LIN {X 0,Y 233.528,Z 742.542,A -85,B 0,C 180,E1 -20220.879,E2 -20220.879} C_VEL
LIN {X 0,Y 229.951,Z 751.909,A -85,B 0,C 180,E1 -20223.691,E2 -20223.691} C_VEL
LIN {X 0,Y 226.657,Z 760.086,A -85,B 0,C 180,E1 -20226.71,E2 -20226.71} C_VEL
LIN {X 0,Y 223.402,Z 768.26,A -85,B 0,C 180,E1 -20230.537,E2 -20230.537} C_VEL
LIN {X 0,Y 221.193,Z 774.434,A -85,B 0,C 180,E1 -20234.329,E2 -20234.329} C_VEL
LIN {X 0,Y 219.975,Z 777.913,A -85,B 0,C 180,E1 -20237.074,E2 -20237.074} C_VEL
LIN {X 0,Y 219.07,Z 781.444,A -85,B 0,C 180,E1 -20240.767,E2 -20240.767} C_VEL
LIN {X 0,Y 218.596,Z 783.762,A -85,B 0,C 180,E1 -20244.462,E2 -20244.462} C_VEL
LIN {X 0,Y 218.545,Z 784.923,A -85,B 0,C 180,E1 -20248.154,E2 -20248.154} C_VEL
LIN {X 0,Y 218.609,Z 785.073,A -85,B 0,C 180,E1 -20249.997,E2 -20249.997} C_VEL
LIN {X 0,Y 218.516,Z 784.473,A -85,B 0,C 180,E1 -20253.685,E2 -20253.685} C_VEL
LIN {X 0,Y 218.782,Z 782.724,A -85,B 0,C 180,E1 -20257.38,E2 -20257.38} C_VEL
LIN {X 0,Y 219.453,Z 779.797,A -85,B 0,C 180,E1 -20261.075,E2 -20261.075} C_VEL
LIN {X 0,Y 220.755,Z 775.622,A -85,B 0,C 180,E1 -20264.752,E2 -20264.752} C_VEL
LIN {X 0,Y 222.669,Z 770.085,A -85,B 0,C 180,E1 -20268.395,E2 -20268.395} C_VEL
LIN {X 0,Y 225.394,Z 763.035,A -85,B 0,C 180,E1 -20271.97,E2 -20271.97} C_VEL
LIN {X 0,Y 228.381,Z 755.478,A -85,B 0,C 180,E1 -20275.029,E2 -20275.029} C_VEL
LIN {X 0,Y 232.043,Z 746.367,A -85,B 0,C 180,E1 -20277.996,E2 -20277.996} C_VEL
LIN {X 0,Y 234.081,Z 740.636,A -85,B 0,C 180,E1 -20279.593,E2 -20279.593} C_VEL
LIN {X 0,Y 238.094,Z 729.914,A -85,B 0,C 180,E1 -20282.091,E2 -20282.091} C_VEL
LIN {X 0,Y 241.988,Z 718.591,A -85,B 0,C 180,E1 -20284.239,E2 -20284.239} C_VEL
LIN {X 0,Y 245.782,Z 706.267,A -85,B 0,C 180,E1 -20286.136,E2 -20286.136} C_VEL
LIN {X 0,Y 249.355,Z 692.827,A -85,B 0,C 180,E1 -20287.794,E2 -20287.794} C_VEL
LIN {X 0,Y 252.492,Z 678.754,A -85,B 0,C 180,E1 -20289.157,E2 -20289.157} C_VEL
LIN {X 0,Y 255.128,Z 664.35,A -85,B 0,C 180,E1 -20290.209,E2 -20290.209} C_VEL
LIN {X 0,Y 257.197,Z 649.607,A -85,B 0,C 180,E1 -20290.977,E2 -20290.977} C_VEL
LIN {X 0,Y 258.499,Z 634.567,A -85,B 0,C 180,E1 -20291.502,E2 -20291.502} C_VEL
LIN {X 0,Y 263.547,Z 543.737,A -85,B 0,C 180,E1 -20293.808,E2 -20293.808} C_VEL
LIN {X 0,Y 264.694,Z 520.773,A -85,B 0,C 180,E1 -20294.417,E2 -20294.417} C_VEL
LIN {X 0,Y 262.231,Z 488.936,A -85,B 0,C 180,E1 -20296.168,E2 -20296.168} C_VEL
LIN {X 0,Y 261.527,Z 482.024,A -85,B 0,C 180,E1 -20296.6,E2 -20296.6} C_VEL
LIN {X 0,Y 255.769,Z 467.358,A -85,B 0,C 180,E1 -20298.63,E2 -20298.63} C_VEL
LIN {X 0,Y 252.814,Z 454.44,A -85,B 0,C 180,E1 -20301.282,E2 -20301.282} C_VEL
LIN {X 0,Y 246.295,Z 442.759,A -85,B 0,C 180,E1 -20305.201,E2 -20305.201} C_VEL
LIN {X 0,Y 241.55,Z 434.953,A -85,B 0,C 180,E1 -20308.418,E2 -20308.418} C_VEL
LIN {X 0,Y 237.263,Z 428.355,A -85,B 0,C 180,E1 -20311.71,E2 -20311.71} C_VEL
LIN {X 0,Y 234.857,Z 424.476,A -85,B 0,C 180,E1 -20313.855,E2 -20313.855} C_VEL
LIN {X 0,Y 231.096,Z 418.944,A -85,B 0,C 180,E1 -20317.658,E2 -20317.658} C_VEL
LIN {X 0,Y 227.762,Z 414.114,A -85,B 0,C 180,E1 -20322.027,E2 -20322.027} C_VEL
LIN {X 0,Y 225.036,Z 409.874,A -85,B 0,C 180,E1 -20327.373,E2 -20327.373} C_VEL
LIN {X 0,Y 224.468,Z 408.787,A -85,B 0,C 180,E1 -20329.172,E2 -20329.172} C_VEL
LIN {X 0,Y 223.393,Z 407.788,A -85,B 0,C 180,E1 -20332.771,E2 -20332.771} C_VEL
LIN {X 0,Y 223.058,Z 407.195,A -85,B 0,C 180,E1 -20338.195,E2 -20338.195} C_VEL
LIN {X 0,Y 223.56,Z 407.709,A -85,B 0,C 180,E1 -20341.802,E2 -20341.802} C_VEL
LIN {X 0,Y 224.445,Z 408.865,A -85,B 0,C 180,E1 -20345.39,E2 -20345.39} C_VEL
LIN {X 0,Y 224.978,Z 409.897,A -85,B 0,C 180,E1 -20347.178,E2 -20347.178} C_VEL
LIN {X 0,Y 227.491,Z 413.981,A -85,B 0,C 180,E1 -20352.489,E2 -20352.489} C_VEL
LIN {X 0,Y 230.597,Z 419.999,A -85,B 0,C 180,E1 -20357.745,E2 -20357.745} C_VEL
LIN {X 0,Y 232.856,Z 424.053,A -85,B 0,C 180,E1 -20360.679,E2 -20360.679} C_VEL
LIN {X 0,Y 236.167,Z 430.465,A -85,B 0,C 180,E1 -20364.622,E2 -20364.622} C_VEL
LIN {X 0,Y 240.43,Z 439.684,A -85,B 0,C 180,E1 -20369.268,E2 -20369.268} C_VEL
LIN {X 0,Y 243.836,Z 447.928,A -85,B 0,C 180,E1 -20372.713,E2 -20372.713} C_VEL
LIN {X 0,Y 247.713,Z 458.603,A -85,B 0,C 180,E1 -20376.57,E2 -20376.57} C_VEL
LIN {X 0,Y 251.328,Z 470.03,A -85,B 0,C 180,E1 -20380.093,E2 -20380.093} C_VEL
LIN {X 0,Y 258.416,Z 484.117,A -85,B 0,C 180,E1 -20382.519,E2 -20382.519} C_VEL
LIN {X 0,Y 261.247,Z 490.693,A -85,B 0,C 180,E1 -20383.447,E2 -20383.447} C_VEL
LIN {X 0,Y 264.994,Z 526.13,A -85,B 0,C 180,E1 -20385.623,E2 -20385.623} C_VEL
LIN {X 0,Y 260.044,Z 616.993,A -85,B 0,C 180,E1 -20387.957,E2 -20387.957} C_VEL
LIN {X 0,Y 258.343,Z 643.193,A -85,B 0,C 180,E1 -20388.662,E2 -20388.662} C_VEL
LIN {X 0,Y 256.535,Z 658.563,A -85,B 0,C 180,E1 -20389.349,E2 -20389.349} C_VEL
LIN {X 0,Y 253.919,Z 673.944,A -85,B 0,C 180,E1 -20390.337,E2 -20390.337} C_VEL
LIN {X 0,Y 251.077,Z 687.643,A -85,B 0,C 180,E1 -20391.534,E2 -20391.534} C_VEL
LIN {X 0,Y 247.46,Z 702.097,A -85,B 0,C 180,E1 -20393.17,E2 -20393.17} C_VEL
LIN {X 0,Y 243.575,Z 715.08,A -85,B 0,C 180,E1 -20395.012,E2 -20395.012} C_VEL
LIN {X 0,Y 239.575,Z 727.078,A -85,B 0,C 180,E1 -20397.136,E2 -20397.136} C_VEL
LIN {X 0,Y 235.608,Z 738.04,A -85,B 0,C 180,E1 -20399.533,E2 -20399.533} C_VEL
LIN {X 0,Y 231.647,Z 748.68,A -85,B 0,C 180,E1 -20402.444,E2 -20402.444} C_VEL
LIN {X 0,Y 228.007,Z 757.529,A -85,B 0,C 180,E1 -20405.414,E2 -20405.414} C_VEL
LIN {X 0,Y 224.702,Z 765.804,A -85,B 0,C 180,E1 -20408.922,E2 -20408.922} C_VEL
LIN {X 0,Y 222.184,Z 772.445,A -85,B 0,C 180,E1 -20412.516,E2 -20412.516} C_VEL
LIN {X 0,Y 220.343,Z 777.639,A -85,B 0,C 180,E1 -20416.163,E2 -20416.163} C_VEL
LIN {X 0,Y 219.41,Z 780.621,A -85,B 0,C 180,E1 -20418.923,E2 -20418.923} C_VEL
LIN {X 0,Y 218.683,Z 783.554,A -85,B 0,C 180,E1 -20422.617,E2 -20422.617} C_VEL
LIN {X 0,Y 218.449,Z 785.315,A -85,B 0,C 180,E1 -20426.314,E2 -20426.314} C_VEL
LIN {X 0,Y 218.487,Z 785.925,A -85,B 0,C 180,E1 -20430.003,E2 -20430.003} C_VEL
LIN {X 0,Y 218.451,Z 785.35,A -85,B 0,C 180,E1 -20433.692,E2 -20433.692} C_VEL
LIN {X 0,Y 218.686,Z 783.636,A -85,B 0,C 180,E1 -20437.389,E2 -20437.389} C_VEL
LIN {X 0,Y 219.405,Z 780.744,A -85,B 0,C 180,E1 -20441.084,E2 -20441.084} C_VEL
LIN {X 0,Y 220.736,Z 776.608,A -85,B 0,C 180,E1 -20444.759,E2 -20444.759} C_VEL
LIN {X 0,Y 222.712,Z 771.129,A -85,B 0,C 180,E1 -20448.398,E2 -20448.398} C_VEL
LIN {X 0,Y 225.381,Z 764.155,A -85,B 0,C 180,E1 -20451.977,E2 -20451.977} C_VEL
LIN {X 0,Y 228.357,Z 756.678,A -85,B 0,C 180,E1 -20455.038,E2 -20455.038} C_VEL
LIN {X 0,Y 232.057,Z 747.668,A -85,B 0,C 180,E1 -20458,E2 -20458} C_VEL
LIN {X 0,Y 235.499,Z 738.47,A -85,B 0,C 180,E1 -20460.489,E2 -20460.489} C_VEL
LIN {X 0,Y 239.814,Z 726.618,A -85,B 0,C 180,E1 -20463.084,E2 -20463.084} C_VEL
LIN {X 0,Y 243.803,Z 714.525,A -85,B 0,C 180,E1 -20465.21,E2 -20465.21} C_VEL
LIN {X 0,Y 247.963,Z 700.812,A -85,B 0,C 180,E1 -20467.108,E2 -20467.108} C_VEL
LIN {X 0,Y 251.05,Z 688.221,A -85,B 0,C 180,E1 -20468.529,E2 -20468.529} C_VEL
LIN {X 0,Y 254.026,Z 673.991,A -85,B 0,C 180,E1 -20469.778,E2 -20469.778} C_VEL
LIN {X 0,Y 256.652,Z 658.624,A -85,B 0,C 180,E1 -20470.765,E2 -20470.765} C_VEL
LIN {X 0,Y 258.471,Z 643.305,A -85,B 0,C 180,E1 -20471.449,E2 -20471.449} C_VEL
LIN {X 0,Y 260.225,Z 615.372,A -85,B 0,C 180,E1 -20472.209,E2 -20472.209} C_VEL
LIN {X 0,Y 265.128,Z 526.826,A -85,B 0,C 180,E1 -20474.466,E2 -20474.466} C_VEL
LIN {X 0,Y 261.714,Z 493.758,A -85,B 0,C 180,E1 -20476.476,E2 -20476.476} C_VEL
LIN {X 0,Y 261.058,Z 489.796,A -85,B 0,C 180,E1 -20476.782,E2 -20476.782} C_VEL
LIN {X 0,Y 255.085,Z 477.378,A -85,B 0,C 180,E1 -20478.737,E2 -20478.737} C_VEL
LIN {X 0,Y 251.148,Z 469.658,A -85,B 0,C 180,E1 -20480.18,E2 -20480.18} C_VEL
LIN {X 0,Y 248.371,Z 460.391,A -85,B 0,C 180,E1 -20483.036,E2 -20483.036} C_VEL
LIN {X 0,Y 245.282,Z 451.699,A -85,B 0,C 180,E1 -20486.032,E2 -20486.032} C_VEL
LIN {X 0,Y 242.786,Z 452.683,A -85,B 0,C 180,E1 -20486.633,E2 -20486.633} C_VEL
LIN {X 0,Y 240.413,Z 454.892,A -85,B 0,C 180,E1 -20486.916,E2 -20486.916} C_VEL
LIN {X 0,Y 239.117,Z 455.744,A -85,B 0,C 180,E1 -20487.164,E2 -20487.164} C_VEL
LIN {X 0,Y 237.468,Z 456.66,A -85,B 0,C 180,E1 -20487.698,E2 -20487.698} C_VEL
LIN {X 0,Y 236.958,Z 458.291,A -85,B 0,C 180,E1 -20487.984,E2 -20487.984} C_VEL
LIN {X 0,Y 235.516,Z 477.969,A -85,B 0,C 180,E1 -20488.956,E2 -20488.956} C_VEL
LIN {X 0,Y 231.592,Z 543.336,A -85,B 0,C 180,E1 -20492.142,E2 -20492.142} C_VEL
LIN {X 0,Y 231.477,Z 546.573,A -85,B 0,C 180,E1 -20492.319,E2 -20492.319} C_VEL
LIN {X 0,Y 229.849,Z 554.131,A -85,B 0,C 180,E1 -20492.701,E2 -20492.701} C_VEL
LIN {X 0,Y 224.375,Z 568.64,A -85,B 0,C 180,E1 -20493.555,E2 -20493.555} C_VEL
LIN {X 0,Y 222.893,Z 574.117,A -85,B 0,C 180,E1 -20493.992,E2 -20493.992} C_VEL
LIN {X 0,Y 222.631,Z 575.96,A -85,B 0,C 180,E1 -20494.163,E2 -20494.163} C_VEL
LIN {X 0,Y 221.241,Z 591.447,A -85,B 0,C 180,E1 -20495.858,E2 -20495.858} C_VEL
LIN {X 0,Y 219.819,Z 605.709,A -85,B 0,C 180,E1 -20497.831,E2 -20497.831} C_VEL
LIN {X 0,Y 218.247,Z 619.879,A -85,B 0,C 180,E1 -20500.237,E2 -20500.237} C_VEL
LIN {X 0,Y 216.85,Z 632.356,A -85,B 0,C 180,E1 -20502.798,E2 -20502.798} C_VEL
LIN {X 0,Y 215.809,Z 642.883,A -85,B 0,C 180,E1 -20505.381,E2 -20505.381} C_VEL
LIN {X 0,Y 214.963,Z 652.625,A -85,B 0,C 180,E1 -20508.209,E2 -20508.209} C_VEL
LIN {X 0,Y 214.288,Z 662.119,A -85,B 0,C 180,E1 -20511.513,E2 -20511.513} C_VEL
LIN {X 0,Y 213.825,Z 669.895,A -85,B 0,C 180,E1 -20514.814,E2 -20514.814} C_VEL
LIN {X 0,Y 213.954,Z 676.304,A -85,B 0,C 180,E1 -20518.117,E2 -20518.117} C_VEL
LIN {X 0,Y 214.356,Z 680.848,A -85,B 0,C 180,E1 -20520.939,E2 -20520.939} C_VEL
LIN {X 0,Y 215.288,Z 684.464,A -85,B 0,C 180,E1 -20523.743,E2 -20523.743} C_VEL
LIN {X 0,Y 216.97,Z 688.103,A -85,B 0,C 180,E1 -20527.444,E2 -20527.444} C_VEL
LIN {X 0,Y 219.235,Z 690.438,A -85,B 0,C 180,E1 -20531.089,E2 -20531.089} C_VEL
LIN {X 0,Y 222.416,Z 691.467,A -85,B 0,C 180,E1 -20534.642,E2 -20534.642} C_VEL
LIN {X 0,Y 226.389,Z 691.234,A -85,B 0,C 180,E1 -20538.086,E2 -20538.086} C_VEL
LIN {X 0,Y 231.163,Z 689.752,A -85,B 0,C 180,E1 -20541.397,E2 -20541.397} C_VEL
LIN {X 0,Y 236.599,Z 687.063,A -85,B 0,C 180,E1 -20544.573,E2 -20544.573} C_VEL
LIN {X 0,Y 242.848,Z 683.069,A -85,B 0,C 180,E1 -20547.583,E2 -20547.583} C_VEL
LIN {X 0,Y 249.683,Z 677.804,A -85,B 0,C 180,E1 -20550.441,E2 -20550.441} C_VEL
LIN {X 0,Y 257.225,Z 671.101,A -85,B 0,C 180,E1 -20553.123,E2 -20553.123} C_VEL
LIN {X 0,Y 266.468,Z 661.723,A -85,B 0,C 180,E1 -20555.933,E2 -20555.933} C_VEL
LIN {X 0,Y 274.167,Z 652.937,A -85,B 0,C 180,E1 -20557.967,E2 -20557.967} C_VEL
LIN {X 0,Y 282.318,Z 642.553,A -85,B 0,C 180,E1 -20559.868,E2 -20559.868} C_VEL
LIN {X 0,Y 289.883,Z 631.739,A -85,B 0,C 180,E1 -20561.455,E2 -20561.455} C_VEL
LIN {X 0,Y 290.674,Z 630.728,A -85,B 0,C 180,E1 -20561.969,E2 -20561.969} C_VEL
LIN {X 0,Y 282.496,Z 644.25,A -85,B 0,C 180,E1 -20563.044,E2 -20563.044} C_VEL
LIN {X 0,Y 273.217,Z 658.093,A -85,B 0,C 180,E1 -20564.451,E2 -20564.451} C_VEL
LIN {X 0,Y 263.853,Z 670.906,A -85,B 0,C 180,E1 -20566.166,E2 -20566.166} C_VEL
LIN {X 0,Y 255.167,Z 682.045,A -85,B 0,C 180,E1 -20568.091,E2 -20568.091} C_VEL
LIN {X 0,Y 246.17,Z 693.075,A -85,B 0,C 180,E1 -20570.561,E2 -20570.561} C_VEL
LIN {X 0,Y 242.773,Z 697.405,A -85,B 0,C 180,E1 -20571.679,E2 -20571.679} C_VEL
LIN {X 0,Y 238.926,Z 710.408,A -85,B 0,C 180,E1 -20573.438,E2 -20573.438} C_VEL
LIN {X 0,Y 235.076,Z 722.055,A -85,B 0,C 180,E1 -20575.384,E2 -20575.384} C_VEL
LIN {X 0,Y 230.719,Z 733.744,A -85,B 0,C 180,E1 -20577.784,E2 -20577.784} C_VEL
LIN {X 0,Y 226.879,Z 743.563,A -85,B 0,C 180,E1 -20580.286,E2 -20580.286} C_VEL
LIN {X 0,Y 223.587,Z 751.929,A -85,B 0,C 180,E1 -20582.882,E2 -20582.882} C_VEL
LIN {X 0,Y 220.096,Z 760.104,A -85,B 0,C 180,E1 -20585.973,E2 -20585.973} C_VEL
LIN {X 0,Y 217.249,Z 766.855,A -85,B 0,C 180,E1 -20589.152,E2 -20589.152} C_VEL
LIN {X 0,Y 214.769,Z 773.102,A -85,B 0,C 180,E1 -20592.869,E2 -20592.869} C_VEL
LIN {X 0,Y 213.011,Z 777.928,A -85,B 0,C 180,E1 -20596.644,E2 -20596.644} C_VEL
LIN {X 0,Y 212.035,Z 781.459,A -85,B 0,C 180,E1 -20600.458,E2 -20600.458} C_VEL
LIN {X 0,Y 211.509,Z 783.777,A -85,B 0,C 180,E1 -20604.276,E2 -20604.276} C_VEL
LIN {X 0,Y 211.447,Z 784.937,A -85,B 0,C 180,E1 -20608.092,E2 -20608.092} C_VEL
LIN {X 0,Y 211.508,Z 785.087,A -85,B 0,C 180,E1 -20609.997,E2 -20609.997} C_VEL
LIN {X 0,Y 211.435,Z 784.487,A -85,B 0,C 180,E1 -20613.809,E2 -20613.809} C_VEL
LIN {X 0,Y 211.705,Z 782.737,A -85,B 0,C 180,E1 -20617.628,E2 -20617.628} C_VEL
LIN {X 0,Y 212.429,Z 779.811,A -85,B 0,C 180,E1 -20621.446,E2 -20621.446} C_VEL
LIN {X 0,Y 213.834,Z 775.635,A -85,B 0,C 180,E1 -20625.241,E2 -20625.241} C_VEL
LIN {X 0,Y 215.871,Z 770.099,A -85,B 0,C 180,E1 -20628.996,E2 -20628.996} C_VEL
LIN {X 0,Y 218.78,Z 763.049,A -85,B 0,C 180,E1 -20632.67,E2 -20632.67} C_VEL
LIN {X 0,Y 221.906,Z 755.493,A -85,B 0,C 180,E1 -20635.812,E2 -20635.812} C_VEL
LIN {X 0,Y 225.736,Z 746.401,A -85,B 0,C 180,E1 -20638.844,E2 -20638.844} C_VEL
LIN {X 0,Y 227.915,Z 740.652,A -85,B 0,C 180,E1 -20640.477,E2 -20640.477} C_VEL
LIN {X 0,Y 232.079,Z 729.932,A -85,B 0,C 180,E1 -20643.027,E2 -20643.027} C_VEL
LIN {X 0,Y 236.138,Z 718.611,A -85,B 0,C 180,E1 -20645.211,E2 -20645.211} C_VEL
LIN {X 0,Y 240.076,Z 706.289,A -85,B 0,C 180,E1 -20647.137,E2 -20647.137} C_VEL
LIN {X 0,Y 243.795,Z 692.779,A -85,B 0,C 180,E1 -20648.826,E2 -20648.826} C_VEL
LIN {X 0,Y 247.025,Z 678.786,A -85,B 0,C 180,E1 -20650.197,E2 -20650.197} C_VEL
LIN {X 0,Y 249.754,Z 664.392,A -85,B 0,C 180,E1 -20651.26,E2 -20651.26} C_VEL
LIN {X 0,Y 251.879,Z 649.667,A -85,B 0,C 180,E1 -20652.036,E2 -20652.036} C_VEL
LIN {X 0,Y 253.227,Z 634.662,A -85,B 0,C 180,E1 -20652.567,E2 -20652.567} C_VEL
LIN {X 0,Y 258.201,Z 548.714,A -85,B 0,C 180,E1 -20654.77,E2 -20654.77} C_VEL
LIN {X 0,Y 259.642,Z 521.952,A -85,B 0,C 180,E1 -20655.478,E2 -20655.478} C_VEL
LIN {X 0,Y 257.4,Z 491.022,A -85,B 0,C 180,E1 -20657.22,E2 -20657.22} C_VEL
LIN {X 0,Y 256.913,Z 485.241,A -85,B 0,C 180,E1 -20657.573,E2 -20657.573} C_VEL
LIN {X 0,Y 250.105,Z 467.63,A -85,B 0,C 180,E1 -20660.097,E2 -20660.097} C_VEL
LIN {X 0,Y 248.118,Z 458.805,A -85,B 0,C 180,E1 -20662.022,E2 -20662.022} C_VEL
LIN {X 0,Y 241.566,Z 446.932,A -85,B 0,C 180,E1 -20666.172,E2 -20666.172} C_VEL
LIN {X 0,Y 236.68,Z 438.97,A -85,B 0,C 180,E1 -20669.682,E2 -20669.682} C_VEL
LIN {X 0,Y 233.538,Z 434.085,A -85,B 0,C 180,E1 -20672.196,E2 -20672.196} C_VEL
LIN {X 0,Y 230.726,Z 429.704,A -85,B 0,C 180,E1 -20674.758,E2 -20674.758} C_VEL
LIN {X 0,Y 227.549,Z 424.802,A -85,B 0,C 180,E1 -20678.246,E2 -20678.246} C_VEL
LIN {X 0,Y 224.875,Z 420.876,A -85,B 0,C 180,E1 -20681.788,E2 -20681.788} C_VEL
LIN {X 0,Y 221.498,Z 415.337,A -85,B 0,C 180,E1 -20689.025,E2 -20689.025} C_VEL
LIN {X 0,Y 220.316,Z 414.179,A -85,B 0,C 180,E1 -20692.669,E2 -20692.669} C_VEL
LIN {X 0,Y 219.848,Z 413.525,A -85,B 0,C 180,E1 -20698.168,E2 -20698.168} C_VEL
LIN {X 0,Y 220.348,Z 414.041,A -85,B 0,C 180,E1 -20701.828,E2 -20701.828} C_VEL
LIN {X 0,Y 221.141,Z 415.225,A -85,B 0,C 180,E1 -20705.471,E2 -20705.471} C_VEL
LIN {X 0,Y 222.959,Z 419.024,A -85,B 0,C 180,E1 -20710.902,E2 -20710.902} C_VEL
LIN {X 0,Y 223.974,Z 420.496,A -85,B 0,C 180,E1 -20712.689,E2 -20712.689} C_VEL
LIN {X 0,Y 226.542,Z 425.419,A -85,B 0,C 180,E1 -20717.141,E2 -20717.141} C_VEL
LIN {X 0,Y 228.829,Z 429.811,A -85,B 0,C 180,E1 -20720.411,E2 -20720.411} C_VEL
LIN {X 0,Y 231.773,Z 435.737,A -85,B 0,C 180,E1 -20724.166,E2 -20724.166} C_VEL
LIN {X 0,Y 235.589,Z 444.131,A -85,B 0,C 180,E1 -20728.51,E2 -20728.51} C_VEL
LIN {X 0,Y 239.217,Z 453.213,A -85,B 0,C 180,E1 -20732.423,E2 -20732.423} C_VEL
LIN {X 0,Y 242.983,Z 463.997,A -85,B 0,C 180,E1 -20736.365,E2 -20736.365} C_VEL
LIN {X 0,Y 245.182,Z 470.656,A -85,B 0,C 180,E1 -20738.424,E2 -20738.424} C_VEL
LIN {X 0,Y 250.91,Z 481.609,A -85,B 0,C 180,E1 -20740.515,E2 -20740.515} C_VEL
LIN {X 0,Y 256.467,Z 493.449,A -85,B 0,C 180,E1 -20742.425,E2 -20742.425} C_VEL
LIN {X 0,Y 259.882,Z 526.978,A -85,B 0,C 180,E1 -20744.547,E2 -20744.547} C_VEL
LIN {X 0,Y 255.609,Z 603.178,A -85,B 0,C 180,E1 -20746.535,E2 -20746.535} C_VEL
LIN {X 0,Y 253.172,Z 641.763,A -85,B 0,C 180,E1 -20747.557,E2 -20747.557} C_VEL
LIN {X 0,Y 251.447,Z 656.811,A -85,B 0,C 180,E1 -20748.211,E2 -20748.211} C_VEL
LIN {X 0,Y 248.96,Z 671.499,A -85,B 0,C 180,E1 -20749.117,E2 -20749.117} C_VEL
LIN {X 0,Y 246.075,Z 685.31,A -85,B 0,C 180,E1 -20750.284,E2 -20750.284} C_VEL
LIN {X 0,Y 242.789,Z 698.47,A -85,B 0,C 180,E1 -20751.714,E2 -20751.714} C_VEL
LIN {X 0,Y 238.969,Z 711.329,A -85,B 0,C 180,E1 -20753.452,E2 -20753.452} C_VEL
LIN {X 0,Y 234.668,Z 723.957,A -85,B 0,C 180,E1 -20755.582,E2 -20755.582} C_VEL
LIN {X 0,Y 230.806,Z 734.534,A -85,B 0,C 180,E1 -20757.804,E2 -20757.804} C_VEL
LIN {X 0,Y 227.023,Z 744.326,A -85,B 0,C 180,E1 -20760.313,E2 -20760.313} C_VEL
LIN {X 0,Y 223.629,Z 752.672,A -85,B 0,C 180,E1 -20762.894,E2 -20762.894} C_VEL
LIN {X 0,Y 220.109,Z 760.826,A -85,B 0,C 180,E1 -20765.98,E2 -20765.98} C_VEL
LIN {X 0,Y 217.277,Z 767.581,A -85,B 0,C 180,E1 -20769.161,E2 -20769.161} C_VEL
LIN {X 0,Y 214.807,Z 773.843,A -85,B 0,C 180,E1 -20772.878,E2 -20772.878} C_VEL
LIN {X 0,Y 212.985,Z 778.68,A -85,B 0,C 180,E1 -20776.648,E2 -20776.648} C_VEL
LIN {X 0,Y 211.963,Z 782.224,A -85,B 0,C 180,E1 -20780.46,E2 -20780.46} C_VEL
LIN {X 0,Y 211.43,Z 784.565,A -85,B 0,C 180,E1 -20784.28,E2 -20784.28} C_VEL
LIN {X 0,Y 211.355,Z 785.754,A -85,B 0,C 180,E1 -20788.097,E2 -20788.097} C_VEL
LIN {X 0,Y 211.391,Z 785.911,A -85,B 0,C 180,E1 -20790.003,E2 -20790.003} C_VEL
LIN {X 0,Y 211.338,Z 785.308,A -85,B 0,C 180,E1 -20793.93,E2 -20793.93} C_VEL
LIN {X 0,Y 211.625,Z 783.621,A -85,B 0,C 180,E1 -20797.637,E2 -20797.637} C_VEL
LIN {X 0,Y 212.387,Z 780.728,A -85,B 0,C 180,E1 -20801.455,E2 -20801.455} C_VEL
LIN {X 0,Y 213.815,Z 776.592,A -85,B 0,C 180,E1 -20805.248,E2 -20805.248} C_VEL
LIN {X 0,Y 215.917,Z 771.113,A -85,B 0,C 180,E1 -20808.998,E2 -20808.998} C_VEL
LIN {X 0,Y 218.767,Z 764.137,A -85,B 0,C 180,E1 -20812.678,E2 -20812.678} C_VEL
LIN {X 0,Y 221.895,Z 756.659,A -85,B 0,C 180,E1 -20815.82,E2 -20815.82} C_VEL
LIN {X 0,Y 225.757,Z 747.647,A -85,B 0,C 180,E1 -20818.853,E2 -20818.853} C_VEL
LIN {X 0,Y 230.023,Z 736.755,A -85,B 0,C 180,E1 -20821.809,E2 -20821.809} C_VEL
LIN {X 0,Y 234.225,Z 725.556,A -85,B 0,C 180,E1 -20824.239,E2 -20824.239} C_VEL
LIN {X 0,Y 238.46,Z 713.252,A -85,B 0,C 180,E1 -20826.382,E2 -20826.382} C_VEL
LIN {X 0,Y 242.534,Z 699.967,A -85,B 0,C 180,E1 -20828.223,E2 -20828.223} C_VEL
LIN {X 0,Y 245.965,Z 686.323,A -85,B 0,C 180,E1 -20829.744,E2 -20829.744} C_VEL
LIN {X 0,Y 248.821,Z 672.79,A -85,B 0,C 180,E1 -20830.917,E2 -20830.917} C_VEL
LIN {X 0,Y 251.439,Z 657.728,A -85,B 0,C 180,E1 -20831.864,E2 -20831.864} C_VEL
LIN {X 0,Y 253.194,Z 643.204,A -85,B 0,C 180,E1 -20832.513,E2 -20832.513} C_VEL
LIN {X 0,Y 255.014,Z 615.219,A -85,B 0,C 180,E1 -20833.281,E2 -20833.281} C_VEL
LIN {X 0,Y 260.029,Z 527.509,A -85,B 0,C 180,E1 -20835.547,E2 -20835.547} C_VEL
LIN {X 0,Y 256.626,Z 493.588,A -85,B 0,C 180,E1 -20837.685,E2 -20837.685} C_VEL
LIN {X 0,Y 251.067,Z 481.846,A -85,B 0,C 180,E1 -20839.594,E2 -20839.594} C_VEL
LIN {X 0,Y 244.774,Z 469.745,A -85,B 0,C 180,E1 -20841.969,E2 -20841.969} C_VEL
LIN {X 0,Y 241.924,Z 460.658,A -85,B 0,C 180,E1 -20844.988,E2 -20844.988} C_VEL
LIN {X 0,Y 241.492,Z 459.436,A -85,B 0,C 180,E1 -20845.424,E2 -20845.424} C_VEL
LIN {X 0,Y 238.773,Z 460.877,A -85,B 0,C 180,E1 -20845.996,E2 -20845.996} C_VEL
LIN {X 0,Y 235.988,Z 462.756,A -85,B 0,C 180,E1 -20846.502,E2 -20846.502} C_VEL
LIN {X 0,Y 233.887,Z 464.895,A -85,B 0,C 180,E1 -20846.71,E2 -20846.71} C_VEL
LIN {X 0,Y 232.162,Z 466.279,A -85,B 0,C 180,E1 -20846.982,E2 -20846.982} C_VEL
LIN {X 0,Y 229.938,Z 467.55,A -85,B 0,C 180,E1 -20847.664,E2 -20847.664} C_VEL
LIN {X 0,Y 229.414,Z 469.317,A -85,B 0,C 180,E1 -20847.97,E2 -20847.97} C_VEL
LIN {X 0,Y 226.327,Z 513.135,A -85,B 0,C 180,E1 -20850.209,E2 -20850.209} C_VEL
LIN {X 0,Y 224.122,Z 553.932,A -85,B 0,C 180,E1 -20852.386,E2 -20852.386} C_VEL
LIN {X 0,Y 223.172,Z 569.704,A -85,B 0,C 180,E1 -20853.588,E2 -20853.588} C_VEL
LIN {X 0,Y 222.631,Z 575.96,A -85,B 0,C 180,E1 -20854.163,E2 -20854.163} C_VEL
LIN {X 0,Y 221.359,Z 581.398,A -85,B 0,C 180,E1 -20854.67,E2 -20854.67} C_VEL
LIN {X 0,Y 214.723,Z 596.806,A -85,B 0,C 180,E1 -20856.321,E2 -20856.321} C_VEL
LIN {X 0,Y 213.252,Z 601.894,A -85,B 0,C 180,E1 -20857.011,E2 -20857.011} C_VEL
LIN {X 0,Y 213.005,Z 603.599,A -85,B 0,C 180,E1 -20857.259,E2 -20857.259} C_VEL
LIN {X 0,Y 211.505,Z 617.468,A -85,B 0,C 180,E1 -20859.58,E2 -20859.58} C_VEL
LIN {X 0,Y 210.012,Z 630.47,A -85,B 0,C 180,E1 -20862.22,E2 -20862.22} C_VEL
LIN {X 0,Y 208.859,Z 641.466,A -85,B 0,C 180,E1 -20864.883,E2 -20864.883} C_VEL
LIN {X 0,Y 207.975,Z 651.587,A -85,B 0,C 180,E1 -20867.807,E2 -20867.807} C_VEL
LIN {X 0,Y 207.257,Z 661.459,A -85,B 0,C 180,E1 -20871.223,E2 -20871.223} C_VEL
LIN {X 0,Y 206.751,Z 669.606,A -85,B 0,C 180,E1 -20874.636,E2 -20874.636} C_VEL
LIN {X 0,Y 206.863,Z 676.329,A -85,B 0,C 180,E1 -20878.053,E2 -20878.053} C_VEL
LIN {X 0,Y 207.251,Z 681.024,A -85,B 0,C 180,E1 -20880.971,E2 -20880.971} C_VEL
LIN {X 0,Y 208.629,Z 686.017,A -85,B 0,C 180,E1 -20884.831,E2 -20884.831} C_VEL
LIN {X 0,Y 209.979,Z 688.828,A -85,B 0,C 180,E1 -20887.694,E2 -20887.694} C_VEL
LIN {X 0,Y 212.357,Z 691.464,A -85,B 0,C 180,E1 -20891.453,E2 -20891.453} C_VEL
LIN {X 0,Y 215.695,Z 692.817,A -85,B 0,C 180,E1 -20895.109,E2 -20895.109} C_VEL
LIN {X 0,Y 219.867,Z 692.915,A -85,B 0,C 180,E1 -20898.641,E2 -20898.641} C_VEL
LIN {X 0,Y 224.852,Z 691.787,A -85,B 0,C 180,E1 -20902.029,E2 -20902.029} C_VEL
LIN {X 0,Y 230.542,Z 689.473,A -85,B 0,C 180,E1 -20905.264,E2 -20905.264} C_VEL
LIN {X 0,Y 237.056,Z 685.892,A -85,B 0,C 180,E1 -20908.317,E2 -20908.317} C_VEL
LIN {X 0,Y 244.16,Z 681.085,A -85,B 0,C 180,E1 -20911.206,E2 -20911.206} C_VEL
LIN {X 0,Y 252.026,Z 674.916,A -85,B 0,C 180,E1 -20913.898,E2 -20913.898} C_VEL
LIN {X 0,Y 260.545,Z 667.288,A -85,B 0,C 180,E1 -20916.401,E2 -20916.401} C_VEL
LIN {X 0,Y 269.565,Z 658.141,A -85,B 0,C 180,E1 -20918.735,E2 -20918.735} C_VEL
LIN {X 0,Y 279.226,Z 647.009,A -85,B 0,C 180,E1 -20920.875,E2 -20920.875} C_VEL
LIN {X 0,Y 280.699,Z 645.242,A -85,B 0,C 180,E1 -20921.167,E2 -20921.167} C_VEL
LIN {X 0,Y 281.704,Z 644.056,A -85,B 0,C 180,E1 -20921.542,E2 -20921.542} C_VEL
LIN {X 0,Y 271.367,Z 658.489,A -85,B 0,C 180,E1 -20922.974,E2 -20922.974} C_VEL
LIN {X 0,Y 261.625,Z 670.884,A -85,B 0,C 180,E1 -20924.61,E2 -20924.61} C_VEL
LIN {X 0,Y 251.341,Z 683.064,A -85,B 0,C 180,E1 -20926.756,E2 -20926.756} C_VEL
LIN {X 0,Y 242.936,Z 692.49,A -85,B 0,C 180,E1 -20928.908,E2 -20928.908} C_VEL
LIN {X 0,Y 236.672,Z 699.518,A -85,B 0,C 180,E1 -20930.872,E2 -20930.872} C_VEL
LIN {X 0,Y 232.388,Z 712.992,A -85,B 0,C 180,E1 -20932.779,E2 -20932.779} C_VEL
LIN {X 0,Y 228.083,Z 725.259,A -85,B 0,C 180,E1 -20934.975,E2 -20934.975} C_VEL
LIN {X 0,Y 223.34,Z 737.263,A -85,B 0,C 180,E1 -20937.657,E2 -20937.657} C_VEL
LIN {X 0,Y 219.54,Z 746.539,A -85,B 0,C 180,E1 -20940.252,E2 -20940.252} C_VEL
LIN {X 0,Y 215.533,Z 755.622,A -85,B 0,C 180,E1 -20943.359,E2 -20943.359} C_VEL
LIN {X 0,Y 212.224,Z 763.159,A -85,B 0,C 180,E1 -20946.582,E2 -20946.582} C_VEL
LIN {X 0,Y 209.127,Z 770.183,A -85,B 0,C 180,E1 -20950.36,E2 -20950.36} C_VEL
LIN {X 0,Y 206.946,Z 775.699,A -85,B 0,C 180,E1 -20954.233,E2 -20954.233} C_VEL
LIN {X 0,Y 205.447,Z 779.865,A -85,B 0,C 180,E1 -20958.153,E2 -20958.153} C_VEL
LIN {X 0,Y 204.656,Z 782.78,A -85,B 0,C 180,E1 -20962.102,E2 -20962.102} C_VEL
LIN {X 0,Y 204.342,Z 784.513,A -85,B 0,C 180,E1 -20966.053,E2 -20966.053} C_VEL
LIN {X 0,Y 204.409,Z 785.101,A -85,B 0,C 180,E1 -20969.997,E2 -20969.997} C_VEL
LIN {X 0,Y 204.324,Z 784.472,A -85,B 0,C 180,E1 -20974.06,E2 -20974.06} C_VEL
LIN {X 0,Y 204.648,Z 782.751,A -85,B 0,C 180,E1 -20977.892,E2 -20977.892} C_VEL
LIN {X 0,Y 205.427,Z 779.824,A -85,B 0,C 180,E1 -20981.842,E2 -20981.842} C_VEL
LIN {X 0,Y 206.937,Z 775.649,A -85,B 0,C 180,E1 -20985.762,E2 -20985.762} C_VEL
LIN {X 0,Y 209.28,Z 769.671,A -85,B 0,C 180,E1 -20989.9,E2 -20989.9} C_VEL
LIN {X 0,Y 212.175,Z 763.064,A -85,B 0,C 180,E1 -20993.417,E2 -20993.417} C_VEL
LIN {X 0,Y 215.491,Z 755.508,A -85,B 0,C 180,E1 -20996.64,E2 -20996.64} C_VEL
LIN {X 0,Y 219.369,Z 746.705,A -85,B 0,C 180,E1 -20999.661,E2 -20999.661} C_VEL
LIN {X 0,Y 221.931,Z 740.346,A -85,B 0,C 180,E1 -21001.497,E2 -21001.497} C_VEL
LIN {X 0,Y 226.144,Z 729.95,A -85,B 0,C 180,E1 -21004.01,E2 -21004.01} C_VEL
LIN {X 0,Y 230.356,Z 718.631,A -85,B 0,C 180,E1 -21006.232,E2 -21006.232} C_VEL
LIN {X 0,Y 234.433,Z 706.312,A -85,B 0,C 180,E1 -21008.189,E2 -21008.189} C_VEL
LIN {X 0,Y 238.179,Z 693.287,A -85,B 0,C 180,E1 -21009.845,E2 -21009.845} C_VEL
LIN {X 0,Y 241.647,Z 678.819,A -85,B 0,C 180,E1 -21011.283,E2 -21011.283} C_VEL
LIN {X 0,Y 244.467,Z 664.435,A -85,B 0,C 180,E1 -21012.356,E2 -21012.356} C_VEL
LIN {X 0,Y 246.774,Z 648.641,A -85,B 0,C 180,E1 -21013.184,E2 -21013.184} C_VEL
LIN {X 0,Y 248.173,Z 633.03,A -85,B 0,C 180,E1 -21013.718,E2 -21013.718} C_VEL
LIN {X 0,Y 253.199,Z 549.164,A -85,B 0,C 180,E1 -21015.89,E2 -21015.89} C_VEL
LIN {X 0,Y 254.661,Z 522.464,A -85,B 0,C 180,E1 -21016.613,E2 -21016.613} C_VEL
LIN {X 0,Y 252.55,Z 491.712,A -85,B 0,C 180,E1 -21018.399,E2 -21018.399} C_VEL
LIN {X 0,Y 252.213,Z 488.11,A -85,B 0,C 180,E1 -21018.638,E2 -21018.638} C_VEL
LIN {X 0,Y 244.491,Z 467.743,A -85,B 0,C 180,E1 -21021.697,E2 -21021.697} C_VEL
LIN {X 0,Y 243.59,Z 463.513,A -85,B 0,C 180,E1 -21022.707,E2 -21022.707} C_VEL
LIN {X 0,Y 237.367,Z 452.102,A -85,B 0,C 180,E1 -21026.787,E2 -21026.787} C_VEL
LIN {X 0,Y 232.876,Z 444.683,A -85,B 0,C 180,E1 -21030.135,E2 -21030.135} C_VEL
LIN {X 0,Y 229.82,Z 439.797,A -85,B 0,C 180,E1 -21032.696,E2 -21032.696} C_VEL
LIN {X 0,Y 227.041,Z 435.434,A -85,B 0,C 180,E1 -21035.299,E2 -21035.299} C_VEL
LIN {X 0,Y 223.968,Z 430.644,A -85,B 0,C 180,E1 -21038.847,E2 -21038.847} C_VEL
LIN {X 0,Y 221.681,Z 427.178,A -85,B 0,C 180,E1 -21041.996,E2 -21041.996} C_VEL
LIN {X 0,Y 218.406,Z 421.873,A -85,B 0,C 180,E1 -21048.868,E2 -21048.868} C_VEL
LIN {X 0,Y 217.233,Z 420.582,A -85,B 0,C 180,E1 -21052.565,E2 -21052.565} C_VEL
LIN {X 0,Y 216.635,Z 419.861,A -85,B 0,C 180,E1 -21058.141,E2 -21058.141} C_VEL
LIN {X 0,Y 217.081,Z 420.368,A -85,B 0,C 180,E1 -21061.855,E2 -21061.855} C_VEL
LIN {X 0,Y 217.836,Z 421.591,A -85,B 0,C 180,E1 -21065.554,E2 -21065.554} C_VEL
LIN {X 0,Y 219.62,Z 425.434,A -85,B 0,C 180,E1 -21071.07,E2 -21071.07} C_VEL
LIN {X 0,Y 220.511,Z 427.01,A -85,B 0,C 180,E1 -21072.891,E2 -21072.891} C_VEL
LIN {X 0,Y 222.998,Z 431.995,A -85,B 0,C 180,E1 -21077.422,E2 -21077.422} C_VEL
LIN {X 0,Y 225.38,Z 436.752,A -85,B 0,C 180,E1 -21080.919,E2 -21080.919} C_VEL
LIN {X 0,Y 227.432,Z 441.052,A -85,B 0,C 180,E1 -21083.686,E2 -21083.686} C_VEL
LIN {X 0,Y 231.158,Z 449.485,A -85,B 0,C 180,E1 -21088.159,E2 -21088.159} C_VEL
LIN {X 0,Y 234.589,Z 458.48,A -85,B 0,C 180,E1 -21092.1,E2 -21092.1} C_VEL
LIN {X 0,Y 238.006,Z 468.483,A -85,B 0,C 180,E1 -21095.808,E2 -21095.808} C_VEL
LIN {X 0,Y 238.891,Z 470.825,A -85,B 0,C 180,E1 -21096.5,E2 -21096.5} C_VEL
LIN {X 0,Y 245.295,Z 482.701,A -85,B 0,C 180,E1 -21099.011,E2 -21099.011} C_VEL
LIN {X 0,Y 251.322,Z 495.48,A -85,B 0,C 180,E1 -21101.217,E2 -21101.217} C_VEL
LIN {X 0,Y 251.992,Z 497.477,A -85,B 0,C 180,E1 -21101.474,E2 -21101.474} C_VEL
LIN {X 0,Y 254.921,Z 529.095,A -85,B 0,C 180,E1 -21103.492,E2 -21103.492} C_VEL
LIN {X 0,Y 248.914,Z 629.281,A -85,B 0,C 180,E1 -21106.095,E2 -21106.095} C_VEL
LIN {X 0,Y 247.521,Z 646.321,A -85,B 0,C 180,E1 -21106.629,E2 -21106.629} C_VEL
LIN {X 0,Y 245.366,Z 662.147,A -85,B 0,C 180,E1 -21107.419,E2 -21107.419} C_VEL
LIN {X 0,Y 242.453,Z 677.161,A -85,B 0,C 180,E1 -21108.469,E2 -21108.469} C_VEL
LIN {X 0,Y 239.026,Z 691.706,A -85,B 0,C 180,E1 -21109.86,E2 -21109.86} C_VEL
LIN {X 0,Y 235.426,Z 704.665,A -85,B 0,C 180,E1 -21111.456,E2 -21111.456} C_VEL
LIN {X 0,Y 231.232,Z 717.348,A -85,B 0,C 180,E1 -21113.386,E2 -21113.386} C_VEL
LIN {X 0,Y 226.974,Z 728.964,A -85,B 0,C 180,E1 -21115.595,E2 -21115.595} C_VEL
LIN {X 0,Y 222.661,Z 739.775,A -85,B 0,C 180,E1 -21118.14,E2 -21118.14} C_VEL
LIN {X 0,Y 219.09,Z 748.649,A -85,B 0,C 180,E1 -21120.716,E2 -21120.716} C_VEL
LIN {X 0,Y 215.052,Z 757.499,A -85,B 0,C 180,E1 -21123.824,E2 -21123.824} C_VEL
LIN {X 0,Y 211.39,Z 765.775,A -85,B 0,C 180,E1 -21127.525,E2 -21127.525} C_VEL
LIN {X 0,Y 208.584,Z 772.417,A -85,B 0,C 180,E1 -21131.335,E2 -21131.335} C_VEL
LIN {X 0,Y 206.482,Z 777.612,A -85,B 0,C 180,E1 -21135.213,E2 -21135.213} C_VEL
LIN {X 0,Y 205.396,Z 780.594,A -85,B 0,C 180,E1 -21138.156,E2 -21138.156} C_VEL
LIN {X 0,Y 204.561,Z 783.527,A -85,B 0,C 180,E1 -21142.104,E2 -21142.104} C_VEL
LIN {X 0,Y 204.256,Z 785.328,A -85,B 0,C 180,E1 -21146.223,E2 -21146.223} C_VEL
LIN {X 0,Y 204.297,Z 785.898,A -85,B 0,C 180,E1 -21150.003,E2 -21150.003} C_VEL
LIN {X 0,Y 204.258,Z 785.322,A -85,B 0,C 180,E1 -21153.949,E2 -21153.949} C_VEL
LIN {X 0,Y 204.563,Z 783.606,A -85,B 0,C 180,E1 -21157.902,E2 -21157.902} C_VEL
LIN {X 0,Y 205.39,Z 780.713,A -85,B 0,C 180,E1 -21161.85,E2 -21161.85} C_VEL
LIN {X 0,Y 206.92,Z 776.576,A -85,B 0,C 180,E1 -21165.769,E2 -21165.769} C_VEL
LIN {X 0,Y 209.35,Z 770.576,A -85,B 0,C 180,E1 -21169.952,E2 -21169.952} C_VEL
LIN {X 0,Y 212.163,Z 764.119,A -85,B 0,C 180,E1 -21173.425,E2 -21173.425} C_VEL
LIN {X 0,Y 215.491,Z 756.64,A -85,B 0,C 180,E1 -21176.647,E2 -21176.647} C_VEL
LIN {X 0,Y 219.459,Z 747.74,A -85,B 0,C 180,E1 -21179.722,E2 -21179.722} C_VEL
LIN {X 0,Y 223.295,Z 738.425,A -85,B 0,C 180,E1 -21182.351,E2 -21182.351} C_VEL
LIN {X 0,Y 227.985,Z 726.568,A -85,B 0,C 180,E1 -21185.043,E2 -21185.043} C_VEL
LIN {X 0,Y 232.327,Z 714.468,A -85,B 0,C 180,E1 -21187.232,E2 -21187.232} C_VEL
LIN {X 0,Y 236.339,Z 702.205,A -85,B 0,C 180,E1 -21188.995,E2 -21188.995} C_VEL
LIN {X 0,Y 239.629,Z 689.869,A -85,B 0,C 180,E1 -21190.461,E2 -21190.461} C_VEL
LIN {X 0,Y 242.799,Z 676.088,A -85,B 0,C 180,E1 -21191.743,E2 -21191.743} C_VEL
LIN {X 0,Y 245.594,Z 661.434,A -85,B 0,C 180,E1 -21192.748,E2 -21192.748} C_VEL
LIN {X 0,Y 247.675,Z 646.364,A -85,B 0,C 180,E1 -21193.484,E2 -21193.484} C_VEL
LIN {X 0,Y 249.023,Z 629.354,A -85,B 0,C 180,E1 -21194.028,E2 -21194.028} C_VEL
LIN {X 0,Y 255.057,Z 529.023,A -85,B 0,C 180,E1 -21196.63,E2 -21196.63} C_VEL
LIN {X 0,Y 252.047,Z 496.89,A -85,B 0,C 180,E1 -21198.695,E2 -21198.695} C_VEL
LIN {X 0,Y 246.462,Z 485.015,A -85,B 0,C 180,E1 -21200.718,E2 -21200.718} C_VEL
LIN {X 0,Y 240.086,Z 472.979,A -85,B 0,C 180,E1 -21203.189,E2 -21203.189} C_VEL
LIN {X 0,Y 238.323,Z 469.431,A -85,B 0,C 180,E1 -21204.041,E2 -21204.041} C_VEL
LIN {X 0,Y 237.688,Z 467.308,A -85,B 0,C 180,E1 -21204.789,E2 -21204.789} C_VEL
LIN {X 0,Y 234.268,Z 469.515,A -85,B 0,C 180,E1 -21205.399,E2 -21205.399} C_VEL
LIN {X 0,Y 231.798,Z 472.261,A -85,B 0,C 180,E1 -21206.042,E2 -21206.042} C_VEL
LIN {X 0,Y 230.618,Z 473.136,A -85,B 0,C 180,E1 -21206.429,E2 -21206.429} C_VEL
LIN {X 0,Y 226.21,Z 488.783,A -85,B 0,C 180,E1 -21207.232,E2 -21207.232} C_VEL
LIN {X 0,Y 223.439,Z 496.717,A -85,B 0,C 180,E1 -21207.875,E2 -21207.875} C_VEL
LIN {X 0,Y 221.475,Z 500.494,A -85,B 0,C 180,E1 -21208.493,E2 -21208.493} C_VEL
LIN {X 0,Y 220.77,Z 502.182,A -85,B 0,C 180,E1 -21208.848,E2 -21208.848} C_VEL
LIN {X 0,Y 219.827,Z 508.88,A -85,B 0,C 180,E1 -21209.486,E2 -21209.486} C_VEL
LIN {X 0,Y 217.844,Z 541.247,A -85,B 0,C 180,E1 -21211.256,E2 -21211.256} C_VEL
LIN {X 0,Y 216.922,Z 559.243,A -85,B 0,C 180,E1 -21212.373,E2 -21212.373} C_VEL
LIN {X 0,Y 215.665,Z 575.741,A -85,B 0,C 180,E1 -21213.805,E2 -21213.805} C_VEL
LIN {X 0,Y 214.265,Z 591.167,A -85,B 0,C 180,E1 -21215.537,E2 -21215.537} C_VEL
LIN {X 0,Y 213.005,Z 603.599,A -85,B 0,C 180,E1 -21217.259,E2 -21217.259} C_VEL
LIN {X 0,Y 211.842,Z 608.676,A -85,B 0,C 180,E1 -21218.009,E2 -21218.009} C_VEL
LIN {X 0,Y 208.165,Z 616.631,A -85,B 0,C 180,E1 -21219.273,E2 -21219.273} C_VEL
LIN {X 0,Y 204.399,Z 624.281,A -85,B 0,C 180,E1 -21220.7,E2 -21220.7} C_VEL
LIN {X 0,Y 203.121,Z 628.887,A -85,B 0,C 180,E1 -21221.689,E2 -21221.689} C_VEL
LIN {X 0,Y 201.94,Z 639.87,A -85,B 0,C 180,E1 -21224.352,E2 -21224.352} C_VEL
LIN {X 0,Y 201,Z 650.375,A -85,B 0,C 180,E1 -21227.377,E2 -21227.377} C_VEL
LIN {X 0,Y 200.206,Z 660.631,A -85,B 0,C 180,E1 -21230.911,E2 -21230.911} C_VEL
LIN {X 0,Y 199.656,Z 669.14,A -85,B 0,C 180,E1 -21234.445,E2 -21234.445} C_VEL
LIN {X 0,Y 199.775,Z 676.146,A -85,B 0,C 180,E1 -21237.984,E2 -21237.984} C_VEL
LIN {X 0,Y 200.153,Z 681.124,A -85,B 0,C 180,E1 -21241.006,E2 -21241.006} C_VEL
LIN {X 0,Y 201.573,Z 686.417,A -85,B 0,C 180,E1 -21245,E2 -21245} C_VEL
LIN {X 0,Y 202.995,Z 689.508,A -85,B 0,C 180,E1 -21247.96,E2 -21247.96} C_VEL
LIN {X 0,Y 205.487,Z 692.456,A -85,B 0,C 180,E1 -21251.842,E2 -21251.842} C_VEL
LIN {X 0,Y 208.981,Z 694.129,A -85,B 0,C 180,E1 -21255.607,E2 -21255.607} C_VEL
LIN {X 0,Y 213.345,Z 694.56,A -85,B 0,C 180,E1 -21259.233,E2 -21259.233} C_VEL
LIN {X 0,Y 218.55,Z 693.789,A -85,B 0,C 180,E1 -21262.699,E2 -21262.699} C_VEL
LIN {X 0,Y 224.497,Z 691.85,A -85,B 0,C 180,E1 -21265.994,E2 -21265.994} C_VEL
LIN {X 0,Y 231.289,Z 688.688,A -85,B 0,C 180,E1 -21269.09,E2 -21269.09} C_VEL
LIN {X 0,Y 238.688,Z 684.35,A -85,B 0,C 180,E1 -21272.005,E2 -21272.005} C_VEL
LIN {X 0,Y 246.852,Z 678.711,A -85,B 0,C 180,E1 -21274.709,E2 -21274.709} C_VEL
LIN {X 0,Y 255.668,Z 671.672,A -85,B 0,C 180,E1 -21277.211,E2 -21277.211} C_VEL
LIN {X 0,Y 264.993,Z 663.188,A -85,B 0,C 180,E1 -21279.532,E2 -21279.532} C_VEL
LIN {X 0,Y 269.921,Z 658.283,A -85,B 0,C 180,E1 -21280.612,E2 -21280.612} C_VEL
LIN {X 0,Y 271.243,Z 657.192,A -85,B 0,C 180,E1 -21281.286,E2 -21281.286} C_VEL
LIN {X 0,Y 261.065,Z 669.363,A -85,B 0,C 180,E1 -21282.81,E2 -21282.81} C_VEL
LIN {X 0,Y 249.675,Z 681.934,A -85,B 0,C 180,E1 -21284.936,E2 -21284.936} C_VEL
LIN {X 0,Y 239.068,Z 692.92,A -85,B 0,C 180,E1 -21287.454,E2 -21287.454} C_VEL
LIN {X 0,Y 230.511,Z 701.729,A -85,B 0,C 180,E1 -21290.043,E2 -21290.043} C_VEL
LIN {X 0,Y 225.913,Z 715.378,A -85,B 0,C 180,E1 -21292.088,E2 -21292.088} C_VEL
LIN {X 0,Y 221.885,Z 726.279,A -85,B 0,C 180,E1 -21294.125,E2 -21294.125} C_VEL
LIN {X 0,Y 217.332,Z 737.285,A -85,B 0,C 180,E1 -21296.648,E2 -21296.648} C_VEL
LIN {X 0,Y 213.222,Z 746.878,A -85,B 0,C 180,E1 -21299.395,E2 -21299.395} C_VEL
LIN {X 0,Y 209.177,Z 755.64,A -85,B 0,C 180,E1 -21302.482,E2 -21302.482} C_VEL
LIN {X 0,Y 205.676,Z 763.177,A -85,B 0,C 180,E1 -21305.789,E2 -21305.789} C_VEL
LIN {X 0,Y 202.393,Z 770.2,A -85,B 0,C 180,E1 -21309.678,E2 -21309.678} C_VEL
LIN {X 0,Y 200.073,Z 775.715,A -85,B 0,C 180,E1 -21313.676,E2 -21313.676} C_VEL
LIN {X 0,Y 198.462,Z 779.88,A -85,B 0,C 180,E1 -21317.73,E2 -21317.73} C_VEL
LIN {X 0,Y 197.596,Z 782.794,A -85,B 0,C 180,E1 -21321.818,E2 -21321.818} C_VEL
LIN {X 0,Y 197.247,Z 784.565,A -85,B 0,C 180,E1 -21326.072,E2 -21326.072} C_VEL
LIN {X 0,Y 197.313,Z 785.115,A -85,B 0,C 180,E1 -21329.997,E2 -21329.997} C_VEL
LIN {X 0,Y 197.245,Z 784.514,A -85,B 0,C 180,E1 -21334.083,E2 -21334.083} C_VEL
LIN {X 0,Y 197.587,Z 782.765,A -85,B 0,C 180,E1 -21338.176,E2 -21338.176} C_VEL
LIN {X 0,Y 198.444,Z 779.838,A -85,B 0,C 180,E1 -21342.265,E2 -21342.265} C_VEL
LIN {X 0,Y 200.064,Z 775.663,A -85,B 0,C 180,E1 -21346.318,E2 -21346.318} C_VEL
LIN {X 0,Y 202.403,Z 770.054,A -85,B 0,C 180,E1 -21350.362,E2 -21350.362} C_VEL
LIN {X 0,Y 205.627,Z 763.078,A -85,B 0,C 180,E1 -21354.21,E2 -21354.21} C_VEL
LIN {X 0,Y 209.138,Z 755.523,A -85,B 0,C 180,E1 -21357.517,E2 -21357.517} C_VEL
LIN {X 0,Y 213.049,Z 747.013,A -85,B 0,C 180,E1 -21360.523,E2 -21360.523} C_VEL
LIN {X 0,Y 215.886,Z 740.363,A -85,B 0,C 180,E1 -21362.486,E2 -21362.486} C_VEL
LIN {X 0,Y 220.285,Z 729.968,A -85,B 0,C 180,E1 -21365.045,E2 -21365.045} C_VEL
LIN {X 0,Y 224.649,Z 718.651,A -85,B 0,C 180,E1 -21367.306,E2 -21367.306} C_VEL
LIN {X 0,Y 228.873,Z 706.335,A -85,B 0,C 180,E1 -21369.292,E2 -21369.292} C_VEL
LIN {X 0,Y 232.881,Z 692.826,A -85,B 0,C 180,E1 -21371.022,E2 -21371.022} C_VEL
LIN {X 0,Y 236.352,Z 678.852,A -85,B 0,C 180,E1 -21372.42,E2 -21372.42} C_VEL
LIN {X 0,Y 239.402,Z 663.732,A -85,B 0,C 180,E1 -21373.544,E2 -21373.544} C_VEL
LIN {X 0,Y 241.651,Z 648.703,A -85,B 0,C 180,E1 -21374.335,E2 -21374.335} C_VEL
LIN {X 0,Y 243.092,Z 633.13,A -85,B 0,C 180,E1 -21374.874,E2 -21374.874} C_VEL
LIN {X 0,Y 248.672,Z 543.035,A -85,B 0,C 180,E1 -21377.235,E2 -21377.235} C_VEL
LIN {X 0,Y 249.839,Z 523.97,A -85,B 0,C 180,E1 -21377.737,E2 -21377.737} C_VEL
LIN {X 0,Y 247.771,Z 491.735,A -85,B 0,C 180,E1 -21379.664,E2 -21379.664} C_VEL
LIN {X 0,Y 242.375,Z 476.751,A -85,B 0,C 180,E1 -21381.897,E2 -21381.897} C_VEL
LIN {X 0,Y 238.985,Z 468.182,A -85,B 0,C 180,E1 -21383.374,E2 -21383.374} C_VEL
LIN {X 0,Y 233.472,Z 457.816,A -85,B 0,C 180,E1 -21387.191,E2 -21387.191} C_VEL
LIN {X 0,Y 229.096,Z 450.377,A -85,B 0,C 180,E1 -21390.605,E2 -21390.605} C_VEL
LIN {X 0,Y 226.111,Z 445.531,A -85,B 0,C 180,E1 -21393.212,E2 -21393.212} C_VEL
LIN {X 0,Y 223.417,Z 441.183,A -85,B 0,C 180,E1 -21395.862,E2 -21395.862} C_VEL
LIN {X 0,Y 220.365,Z 436.445,A -85,B 0,C 180,E1 -21399.463,E2 -21399.463} C_VEL
LIN {X 0,Y 217.827,Z 432.688,A -85,B 0,C 180,E1 -21403.12,E2 -21403.12} C_VEL
LIN {X 0,Y 215.277,Z 428.383,A -85,B 0,C 180,E1 -21408.704,E2 -21408.704} C_VEL
LIN {X 0,Y 214.148,Z 426.992,A -85,B 0,C 180,E1 -21412.457,E2 -21412.457} C_VEL
LIN {X 0,Y 213.512,Z 426.216,A -85,B 0,C 180,E1 -21418.114,E2 -21418.114} C_VEL
LIN {X 0,Y 213.795,Z 426.67,A -85,B 0,C 180,E1 -21421.884,E2 -21421.884} C_VEL
LIN {X 0,Y 214.525,Z 427.959,A -85,B 0,C 180,E1 -21425.64,E2 -21425.64} C_VEL
LIN {X 0,Y 216.229,Z 431.849,A -85,B 0,C 180,E1 -21431.246,E2 -21431.246} C_VEL
LIN {X 0,Y 217.939,Z 435.406,A -85,B 0,C 180,E1 -21434.95,E2 -21434.95} C_VEL
LIN {X 0,Y 220.044,Z 439.666,A -85,B 0,C 180,E1 -21438.626,E2 -21438.626} C_VEL
LIN {X 0,Y 223.177,Z 446.407,A -85,B 0,C 180,E1 -21443.181,E2 -21443.181} C_VEL
LIN {X 0,Y 226.702,Z 454.706,A -85,B 0,C 180,E1 -21447.711,E2 -21447.711} C_VEL
LIN {X 0,Y 229.73,Z 462.816,A -85,B 0,C 180,E1 -21451.337,E2 -21451.337} C_VEL
LIN {X 0,Y 232.314,Z 470.388,A -85,B 0,C 180,E1 -21454.229,E2 -21454.229} C_VEL
LIN {X 0,Y 238.061,Z 480.569,A -85,B 0,C 180,E1 -21456.714,E2 -21456.714} C_VEL
LIN {X 0,Y 243.617,Z 491.773,A -85,B 0,C 180,E1 -21458.942,E2 -21458.942} C_VEL
LIN {X 0,Y 247.436,Z 500.377,A -85,B 0,C 180,E1 -21460.398,E2 -21460.398} C_VEL
LIN {X 0,Y 250.006,Z 530.409,A -85,B 0,C 180,E1 -21462.351,E2 -21462.351} C_VEL
LIN {X 0,Y 243.842,Z 629.179,A -85,B 0,C 180,E1 -21464.937,E2 -21464.937} C_VEL
LIN {X 0,Y 242.408,Z 646.258,A -85,B 0,C 180,E1 -21465.477,E2 -21465.477} C_VEL
LIN {X 0,Y 240.19,Z 662.103,A -85,B 0,C 180,E1 -21466.274,E2 -21466.274} C_VEL
LIN {X 0,Y 237.191,Z 677.128,A -85,B 0,C 180,E1 -21467.333,E2 -21467.333} C_VEL
LIN {X 0,Y 233.922,Z 690.673,A -85,B 0,C 180,E1 -21468.63,E2 -21468.63} C_VEL
LIN {X 0,Y 229.904,Z 704.642,A -85,B 0,C 180,E1 -21470.351,E2 -21470.351} C_VEL
LIN {X 0,Y 225.564,Z 717.328,A -85,B 0,C 180,E1 -21472.309,E2 -21472.309} C_VEL
LIN {X 0,Y 221.109,Z 728.946,A -85,B 0,C 180,E1 -21474.548,E2 -21474.548} C_VEL
LIN {X 0,Y 216.621,Z 739.758,A -85,B 0,C 180,E1 -21477.142,E2 -21477.142} C_VEL
LIN {X 0,Y 212.878,Z 748.652,A -85,B 0,C 180,E1 -21479.782,E2 -21479.782} C_VEL
LIN {X 0,Y 208.639,Z 757.484,A -85,B 0,C 180,E1 -21482.955,E2 -21482.955} C_VEL
LIN {X 0,Y 204.785,Z 765.76,A -85,B 0,C 180,E1 -21486.758,E2 -21486.758} C_VEL
